REGION Network 4: Call production data cycle timer
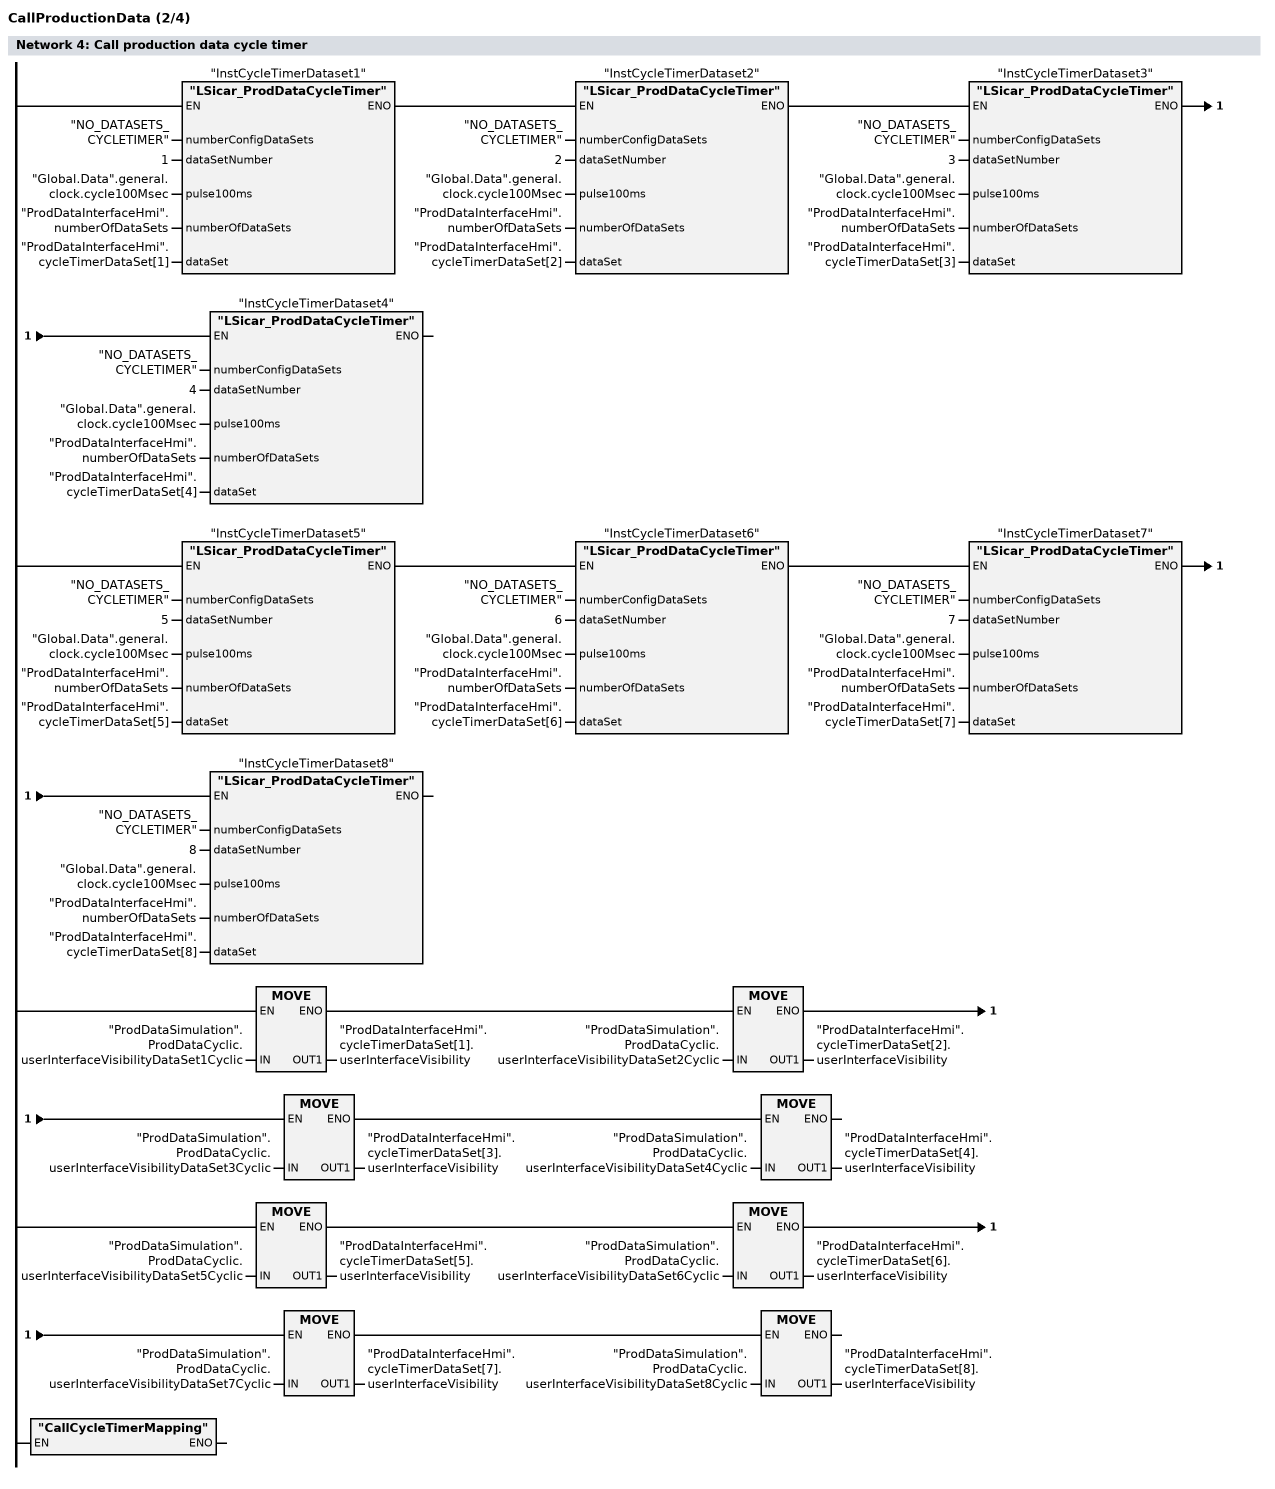
   RUNG wire#powerrail
      "InstCycleTimerDataset1"(numberConfigDataSets := "NO_DATASETS_CYCLETIMER", dataSetNumber := 1, pulse100ms := "Global.Data".general.clock.cycle100Msec, numberOfDataSets := "ProdDataInterfaceHmi".numberOfDataSets, dataSet := "ProdDataInterfaceHmi".cycleTimerDataSet[1])
      "InstCycleTimerDataset2"(numberConfigDataSets := "NO_DATASETS_CYCLETIMER", dataSetNumber := 2, pulse100ms := "Global.Data".general.clock.cycle100Msec, numberOfDataSets := "ProdDataInterfaceHmi".numberOfDataSets, dataSet := "ProdDataInterfaceHmi".cycleTimerDataSet[2])
      "InstCycleTimerDataset3"(numberConfigDataSets := "NO_DATASETS_CYCLETIMER", dataSetNumber := 3, pulse100ms := "Global.Data".general.clock.cycle100Msec, numberOfDataSets := "ProdDataInterfaceHmi".numberOfDataSets, dataSet := "ProdDataInterfaceHmi".cycleTimerDataSet[3])
      "InstCycleTimerDataset4"(numberConfigDataSets := "NO_DATASETS_CYCLETIMER", dataSetNumber := 4, pulse100ms := "Global.Data".general.clock.cycle100Msec, numberOfDataSets := "ProdDataInterfaceHmi".numberOfDataSets, dataSet := "ProdDataInterfaceHmi".cycleTimerDataSet[4])
   END_RUNG
   RUNG wire#powerrail
      "InstCycleTimerDataset5"(numberConfigDataSets := "NO_DATASETS_CYCLETIMER", dataSetNumber := 5, pulse100ms := "Global.Data".general.clock.cycle100Msec, numberOfDataSets := "ProdDataInterfaceHmi".numberOfDataSets, dataSet := "ProdDataInterfaceHmi".cycleTimerDataSet[5])
      "InstCycleTimerDataset6"(numberConfigDataSets := "NO_DATASETS_CYCLETIMER", dataSetNumber := 6, pulse100ms := "Global.Data".general.clock.cycle100Msec, numberOfDataSets := "ProdDataInterfaceHmi".numberOfDataSets, dataSet := "ProdDataInterfaceHmi".cycleTimerDataSet[6])
      "InstCycleTimerDataset7"(numberConfigDataSets := "NO_DATASETS_CYCLETIMER", dataSetNumber := 7, pulse100ms := "Global.Data".general.clock.cycle100Msec, numberOfDataSets := "ProdDataInterfaceHmi".numberOfDataSets, dataSet := "ProdDataInterfaceHmi".cycleTimerDataSet[7])
      "InstCycleTimerDataset8"(numberConfigDataSets := "NO_DATASETS_CYCLETIMER", dataSetNumber := 8, pulse100ms := "Global.Data".general.clock.cycle100Msec, numberOfDataSets := "ProdDataInterfaceHmi".numberOfDataSets, dataSet := "ProdDataInterfaceHmi".cycleTimerDataSet[8])
   END_RUNG
   RUNG wire#powerrail
      Move(in := "ProdDataSimulation".ProdDataCyclic.userInterfaceVisibilityDataSet1Cyclic, out1 => "ProdDataInterfaceHmi".cycleTimerDataSet[1].userInterfaceVisibility)
      Move(in := "ProdDataSimulation".ProdDataCyclic.userInterfaceVisibilityDataSet2Cyclic, out1 => "ProdDataInterfaceHmi".cycleTimerDataSet[2].userInterfaceVisibility)
      Move(in := "ProdDataSimulation".ProdDataCyclic.userInterfaceVisibilityDataSet3Cyclic, out1 => "ProdDataInterfaceHmi".cycleTimerDataSet[3].userInterfaceVisibility)
      Move(in := "ProdDataSimulation".ProdDataCyclic.userInterfaceVisibilityDataSet4Cyclic, out1 => "ProdDataInterfaceHmi".cycleTimerDataSet[4].userInterfaceVisibility)
   END_RUNG
   RUNG wire#powerrail
      Move(in := "ProdDataSimulation".ProdDataCyclic.userInterfaceVisibilityDataSet5Cyclic, out1 => "ProdDataInterfaceHmi".cycleTimerDataSet[5].userInterfaceVisibility)
      Move(in := "ProdDataSimulation".ProdDataCyclic.userInterfaceVisibilityDataSet6Cyclic, out1 => "ProdDataInterfaceHmi".cycleTimerDataSet[6].userInterfaceVisibility)
      Move(in := "ProdDataSimulation".ProdDataCyclic.userInterfaceVisibilityDataSet7Cyclic, out1 => "ProdDataInterfaceHmi".cycleTimerDataSet[7].userInterfaceVisibility)
      Move(in := "ProdDataSimulation".ProdDataCyclic.userInterfaceVisibilityDataSet8Cyclic, out1 => "ProdDataInterfaceHmi".cycleTimerDataSet[8].userInterfaceVisibility)
   END_RUNG
   RUNG wire#powerrail
      "CallCycleTimerMapping"()
   END_RUNG
   // the same network as SCL:
   "InstCycleTimerDataset1"(numberConfigDataSets := "NO_DATASETS_CYCLETIMER",   // "LSicar_ProdDataCycleTimer"
                           dataSetNumber := 1,
                           pulse100ms := "Global.Data".general.clock.cycle100Msec,
                           numberOfDataSets := "ProdDataInterfaceHmi".numberOfDataSets,
                           dataSet := "ProdDataInterfaceHmi".cycleTimerDataSet[1],
                           ENO => #_w1);
   "InstCycleTimerDataset2"(EN := #_w1,   // "LSicar_ProdDataCycleTimer"
                           numberConfigDataSets := "NO_DATASETS_CYCLETIMER",
                           dataSetNumber := 2,
                           pulse100ms := "Global.Data".general.clock.cycle100Msec,
                           numberOfDataSets := "ProdDataInterfaceHmi".numberOfDataSets,
                           dataSet := "ProdDataInterfaceHmi".cycleTimerDataSet[2],
                           ENO => #_w2);
   "InstCycleTimerDataset3"(EN := #_w2,   // "LSicar_ProdDataCycleTimer"
                           numberConfigDataSets := "NO_DATASETS_CYCLETIMER",
                           dataSetNumber := 3,
                           pulse100ms := "Global.Data".general.clock.cycle100Msec,
                           numberOfDataSets := "ProdDataInterfaceHmi".numberOfDataSets,
                           dataSet := "ProdDataInterfaceHmi".cycleTimerDataSet[3],
                           ENO => #_w3);
   IF #_w3 THEN
       "InstCycleTimerDataset4"(numberConfigDataSets := "NO_DATASETS_CYCLETIMER",   // "LSicar_ProdDataCycleTimer"
                               dataSetNumber := 4,
                               pulse100ms := "Global.Data".general.clock.cycle100Msec,
                               numberOfDataSets := "ProdDataInterfaceHmi".numberOfDataSets,
                               dataSet := "ProdDataInterfaceHmi".cycleTimerDataSet[4]);
   END_IF;
   "InstCycleTimerDataset5"(numberConfigDataSets := "NO_DATASETS_CYCLETIMER",   // "LSicar_ProdDataCycleTimer"
                           dataSetNumber := 5,
                           pulse100ms := "Global.Data".general.clock.cycle100Msec,
                           numberOfDataSets := "ProdDataInterfaceHmi".numberOfDataSets,
                           dataSet := "ProdDataInterfaceHmi".cycleTimerDataSet[5],
                           ENO => #_w4);
   "InstCycleTimerDataset6"(EN := #_w4,   // "LSicar_ProdDataCycleTimer"
                           numberConfigDataSets := "NO_DATASETS_CYCLETIMER",
                           dataSetNumber := 6,
                           pulse100ms := "Global.Data".general.clock.cycle100Msec,
                           numberOfDataSets := "ProdDataInterfaceHmi".numberOfDataSets,
                           dataSet := "ProdDataInterfaceHmi".cycleTimerDataSet[6],
                           ENO => #_w5);
   "InstCycleTimerDataset7"(EN := #_w5,   // "LSicar_ProdDataCycleTimer"
                           numberConfigDataSets := "NO_DATASETS_CYCLETIMER",
                           dataSetNumber := 7,
                           pulse100ms := "Global.Data".general.clock.cycle100Msec,
                           numberOfDataSets := "ProdDataInterfaceHmi".numberOfDataSets,
                           dataSet := "ProdDataInterfaceHmi".cycleTimerDataSet[7],
                           ENO => #_w6);
   IF #_w6 THEN
       "InstCycleTimerDataset8"(numberConfigDataSets := "NO_DATASETS_CYCLETIMER",   // "LSicar_ProdDataCycleTimer"
                               dataSetNumber := 8,
                               pulse100ms := "Global.Data".general.clock.cycle100Msec,
                               numberOfDataSets := "ProdDataInterfaceHmi".numberOfDataSets,
                               dataSet := "ProdDataInterfaceHmi".cycleTimerDataSet[8]);
   END_IF;
   "ProdDataInterfaceHmi".cycleTimerDataSet[1].userInterfaceVisibility := "ProdDataSimulation".ProdDataCyclic.userInterfaceVisibilityDataSet1Cyclic;
   "ProdDataInterfaceHmi".cycleTimerDataSet[2].userInterfaceVisibility := "ProdDataSimulation".ProdDataCyclic.userInterfaceVisibilityDataSet2Cyclic;
   "ProdDataInterfaceHmi".cycleTimerDataSet[3].userInterfaceVisibility := "ProdDataSimulation".ProdDataCyclic.userInterfaceVisibilityDataSet3Cyclic;
   "ProdDataInterfaceHmi".cycleTimerDataSet[4].userInterfaceVisibility := "ProdDataSimulation".ProdDataCyclic.userInterfaceVisibilityDataSet4Cyclic;
   "ProdDataInterfaceHmi".cycleTimerDataSet[5].userInterfaceVisibility := "ProdDataSimulation".ProdDataCyclic.userInterfaceVisibilityDataSet5Cyclic;
   "ProdDataInterfaceHmi".cycleTimerDataSet[6].userInterfaceVisibility := "ProdDataSimulation".ProdDataCyclic.userInterfaceVisibilityDataSet6Cyclic;
   "ProdDataInterfaceHmi".cycleTimerDataSet[7].userInterfaceVisibility := "ProdDataSimulation".ProdDataCyclic.userInterfaceVisibilityDataSet7Cyclic;
   "ProdDataInterfaceHmi".cycleTimerDataSet[8].userInterfaceVisibility := "ProdDataSimulation".ProdDataCyclic.userInterfaceVisibilityDataSet8Cyclic;
   "CallCycleTimerMapping"();
END_REGION

REGION Network 5: Beispiel: Limit Value 1..2 / Call production data limit values
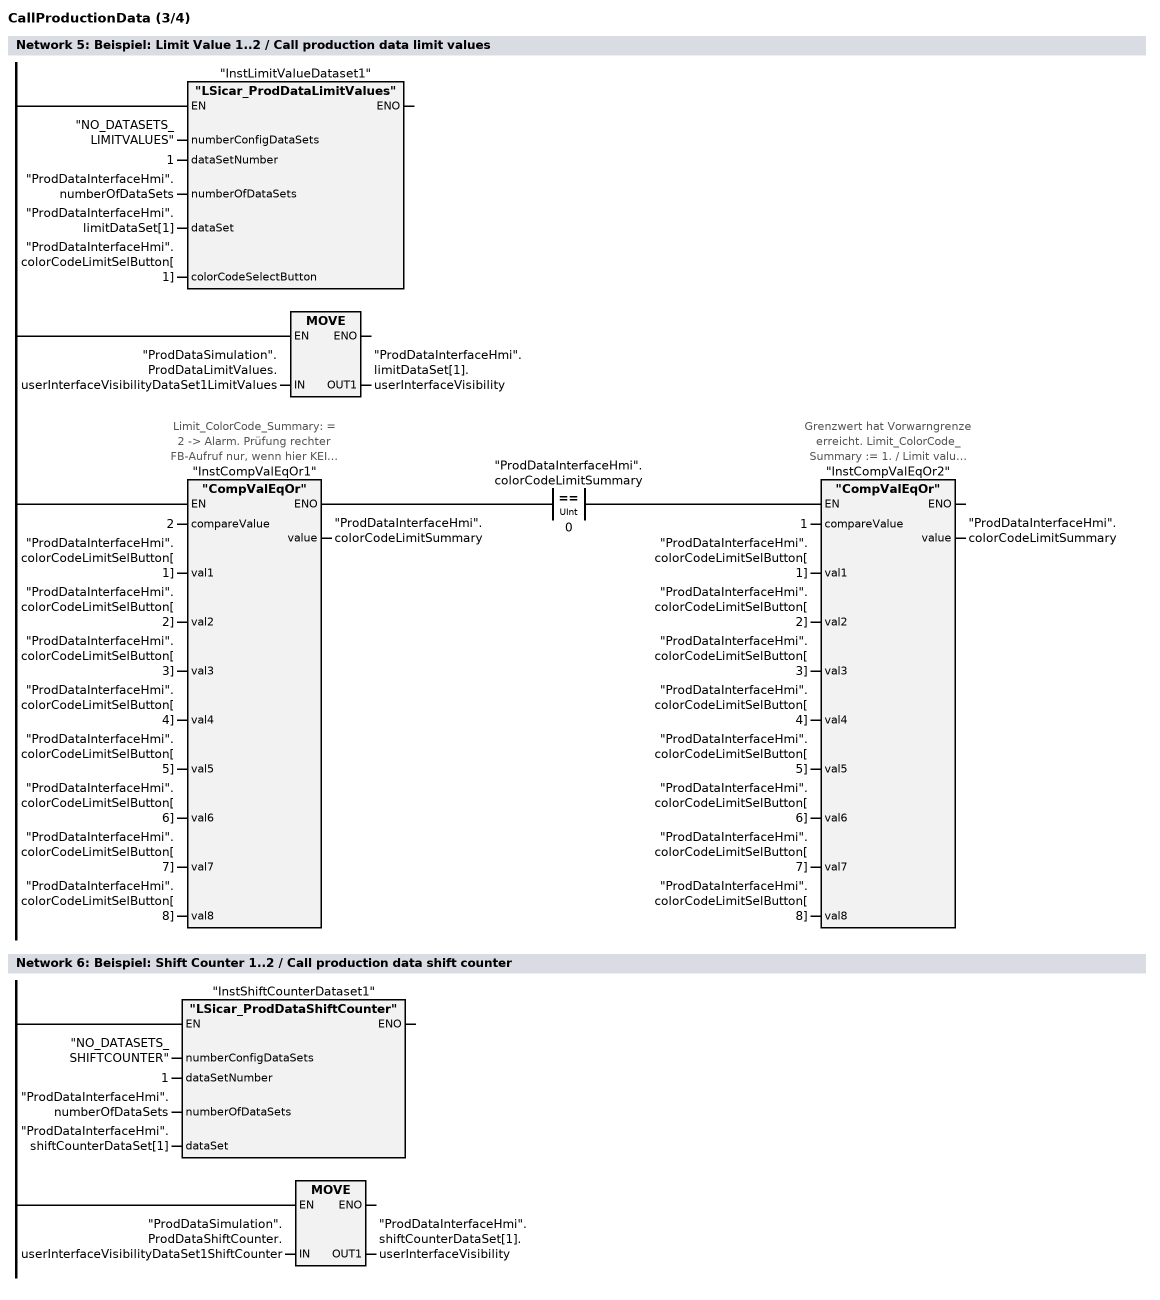
   RUNG wire#powerrail
      "InstLimitValueDataset1"(numberConfigDataSets := "NO_DATASETS_LIMITVALUES", dataSetNumber := 1, numberOfDataSets := "ProdDataInterfaceHmi".numberOfDataSets, dataSet := "ProdDataInterfaceHmi".limitDataSet[1], colorCodeSelectButton := "ProdDataInterfaceHmi".colorCodeLimitSelButton[1])
   END_RUNG
   RUNG wire#powerrail
      Move(in := "ProdDataSimulation".ProdDataLimitValues.userInterfaceVisibilityDataSet1LimitValues, out1 => "ProdDataInterfaceHmi".limitDataSet[1].userInterfaceVisibility)
   END_RUNG
   RUNG wire#powerrail
      "InstCompValEqOr1"(compareValue := 2, val1 := "ProdDataInterfaceHmi".colorCodeLimitSelButton[1], val2 := "ProdDataInterfaceHmi".colorCodeLimitSelButton[2], val3 := "ProdDataInterfaceHmi".colorCodeLimitSelButton[3], val4 := "ProdDataInterfaceHmi".colorCodeLimitSelButton[4], val5 := "ProdDataInterfaceHmi".colorCodeLimitSelButton[5], val6 := "ProdDataInterfaceHmi".colorCodeLimitSelButton[6], val7 := "ProdDataInterfaceHmi".colorCodeLimitSelButton[7], val8 := "ProdDataInterfaceHmi".colorCodeLimitSelButton[8], value => "ProdDataInterfaceHmi".colorCodeLimitSummary)   // Limit_ColorCode_Summary: = 2 -> Alarm. Prüfung rechter FB-Aufruf nur, wenn hier KEIN Alarm (VALUE = 0) ansteht; Alarm ist höher prior. / Limit value = 2 -> Alarm. Limit_ColorCode_Summary := 2. Call right block only, if NO alarm (VALUE = 0) is pending here; alarm is higher prior.
      { S7_Templates := "SrcType := UInt" } EQ_Contact(in1 := "ProdDataInterfaceHmi".colorCodeLimitSummary, in2 := 0)
      "InstCompValEqOr2"(compareValue := 1, val1 := "ProdDataInterfaceHmi".colorCodeLimitSelButton[1], val2 := "ProdDataInterfaceHmi".colorCodeLimitSelButton[2], val3 := "ProdDataInterfaceHmi".colorCodeLimitSelButton[3], val4 := "ProdDataInterfaceHmi".colorCodeLimitSelButton[4], val5 := "ProdDataInterfaceHmi".colorCodeLimitSelButton[5], val6 := "ProdDataInterfaceHmi".colorCodeLimitSelButton[6], val7 := "ProdDataInterfaceHmi".colorCodeLimitSelButton[7], val8 := "ProdDataInterfaceHmi".colorCodeLimitSelButton[8], value => "ProdDataInterfaceHmi".colorCodeLimitSummary)   // Grenzwert hat Vorwarngrenze erreicht. Limit_ColorCode_Summary := 1. / Limit value <= Prewarn value. Limit_ColorCode_Summary := 1.
   END_RUNG
   // the same network as SCL:
   "InstLimitValueDataset1"(numberConfigDataSets := "NO_DATASETS_LIMITVALUES",   // "LSicar_ProdDataLimitValues"
                           dataSetNumber := 1,
                           numberOfDataSets := "ProdDataInterfaceHmi".numberOfDataSets,
                           dataSet := "ProdDataInterfaceHmi".limitDataSet[1],
                           colorCodeSelectButton := "ProdDataInterfaceHmi".colorCodeLimitSelButton[1]);
   "ProdDataInterfaceHmi".limitDataSet[1].userInterfaceVisibility := "ProdDataSimulation".ProdDataLimitValues.userInterfaceVisibilityDataSet1LimitValues;
   "InstCompValEqOr1"(compareValue := 2,   // "CompValEqOr": Limit_ColorCode_Summary: = 2 -> Alarm. Prüfung rechter FB-Aufruf nur, wenn hier KEIN Alarm (VALUE = 0) ansteht; Alarm ist höher prior. / Limit value = 2 -> Alarm. Limit_ColorCode_Summary := 2. Call right block only, if NO alarm (VALUE = 0) is pending here; alarm is higher prior.
                      val1 := "ProdDataInterfaceHmi".colorCodeLimitSelButton[1],
                      val2 := "ProdDataInterfaceHmi".colorCodeLimitSelButton[2],
                      val3 := "ProdDataInterfaceHmi".colorCodeLimitSelButton[3],
                      val4 := "ProdDataInterfaceHmi".colorCodeLimitSelButton[4],
                      val5 := "ProdDataInterfaceHmi".colorCodeLimitSelButton[5],
                      val6 := "ProdDataInterfaceHmi".colorCodeLimitSelButton[6],
                      val7 := "ProdDataInterfaceHmi".colorCodeLimitSelButton[7],
                      val8 := "ProdDataInterfaceHmi".colorCodeLimitSelButton[8],
                      value => "ProdDataInterfaceHmi".colorCodeLimitSummary,
                      ENO => #_w1);
   IF #_w1 AND ("ProdDataInterfaceHmi".colorCodeLimitSummary = 0) THEN
       "InstCompValEqOr2"(compareValue := 1,   // "CompValEqOr": Grenzwert hat Vorwarngrenze erreicht. Limit_ColorCode_Summary := 1. / Limit value <= Prewarn value. Limit_ColorCode_Summary := 1.
                          val1 := "ProdDataInterfaceHmi".colorCodeLimitSelButton[1],
                          val2 := "ProdDataInterfaceHmi".colorCodeLimitSelButton[2],
                          val3 := "ProdDataInterfaceHmi".colorCodeLimitSelButton[3],
                          val4 := "ProdDataInterfaceHmi".colorCodeLimitSelButton[4],
                          val5 := "ProdDataInterfaceHmi".colorCodeLimitSelButton[5],
                          val6 := "ProdDataInterfaceHmi".colorCodeLimitSelButton[6],
                          val7 := "ProdDataInterfaceHmi".colorCodeLimitSelButton[7],
                          val8 := "ProdDataInterfaceHmi".colorCodeLimitSelButton[8],
                          value => "ProdDataInterfaceHmi".colorCodeLimitSummary);
   END_IF;
END_REGION

REGION Network 6: Beispiel: Shift Counter 1..2 / Call production data shift counter
   RUNG wire#powerrail
      "InstShiftCounterDataset1"(numberConfigDataSets := "NO_DATASETS_SHIFTCOUNTER", dataSetNumber := 1, numberOfDataSets := "ProdDataInterfaceHmi".numberOfDataSets, dataSet := "ProdDataInterfaceHmi".shiftCounterDataSet[1])
   END_RUNG
   RUNG wire#powerrail
      Move(in := "ProdDataSimulation".ProdDataShiftCounter.userInterfaceVisibilityDataSet1ShiftCounter, out1 => "ProdDataInterfaceHmi".shiftCounterDataSet[1].userInterfaceVisibility)
   END_RUNG
   // the same network as SCL:
   "InstShiftCounterDataset1"(numberConfigDataSets := "NO_DATASETS_SHIFTCOUNTER",   // "LSicar_ProdDataShiftCounter"
                           dataSetNumber := 1,
                           numberOfDataSets := "ProdDataInterfaceHmi".numberOfDataSets,
                           dataSet := "ProdDataInterfaceHmi".shiftCounterDataSet[1]);
   "ProdDataInterfaceHmi".shiftCounterDataSet[1].userInterfaceVisibility := "ProdDataSimulation".ProdDataShiftCounter.userInterfaceVisibilityDataSet1ShiftCounter;
END_REGION

REGION Network 7: Beispiel Schichtproduktions-Zeiten / Call shift production times
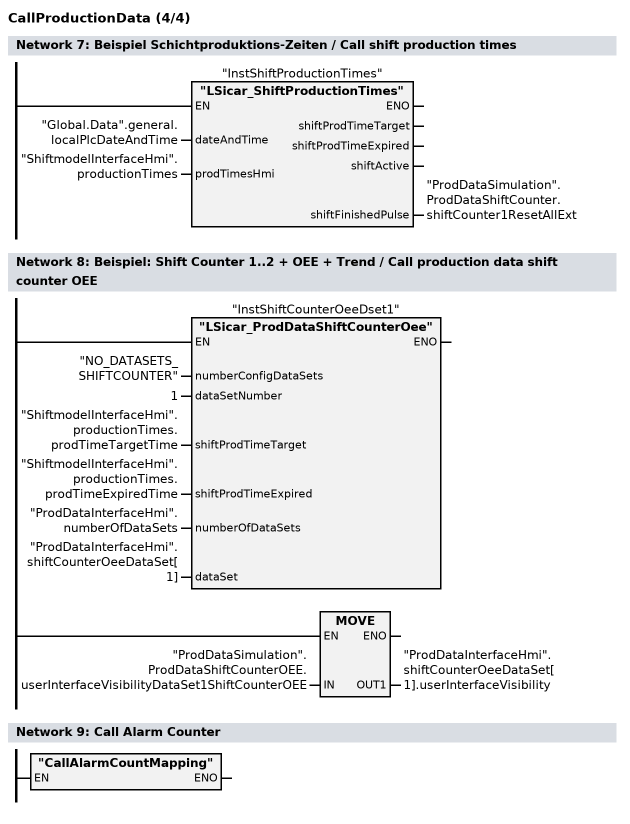
   RUNG wire#powerrail
      "InstShiftProductionTimes"(dateAndTime := "Global.Data".general.localPlcDateAndTime, prodTimesHmi := "ShiftmodelInterfaceHmi".productionTimes, shiftProdTimeTarget =>, shiftProdTimeExpired =>, shiftActive =>, shiftFinishedPulse => "ProdDataSimulation".ProdDataShiftCounter.shiftCounter1ResetAllExt)
   END_RUNG
   // the same network as SCL:
   "InstShiftProductionTimes"(dateAndTime := "Global.Data".general.localPlcDateAndTime,   // "LSicar_ShiftProductionTimes"
                           prodTimesHmi := "ShiftmodelInterfaceHmi".productionTimes,
                           shiftFinishedPulse => "ProdDataSimulation".ProdDataShiftCounter.shiftCounter1ResetAllExt);
END_REGION

REGION Network 8: Beispiel: Shift Counter 1..2 + OEE + Trend / Call production data shift counter OEE
   RUNG wire#powerrail
      "InstShiftCounterOeeDset1"(numberConfigDataSets := "NO_DATASETS_SHIFTCOUNTER", dataSetNumber := 1, shiftProdTimeTarget := "ShiftmodelInterfaceHmi".productionTimes.prodTimeTargetTime, shiftProdTimeExpired := "ShiftmodelInterfaceHmi".productionTimes.prodTimeExpiredTime, numberOfDataSets := "ProdDataInterfaceHmi".numberOfDataSets, dataSet := "ProdDataInterfaceHmi".shiftCounterOeeDataSet[1])
   END_RUNG
   RUNG wire#powerrail
      Move(in := "ProdDataSimulation".ProdDataShiftCounterOEE.userInterfaceVisibilityDataSet1ShiftCounterOEE, out1 => "ProdDataInterfaceHmi".shiftCounterOeeDataSet[1].userInterfaceVisibility)
   END_RUNG
   // the same network as SCL:
   "InstShiftCounterOeeDset1"(numberConfigDataSets := "NO_DATASETS_SHIFTCOUNTER",   // "LSicar_ProdDataShiftCounterOee"
                           dataSetNumber := 1,
                           shiftProdTimeTarget := "ShiftmodelInterfaceHmi".productionTimes.prodTimeTargetTime,
                           shiftProdTimeExpired := "ShiftmodelInterfaceHmi".productionTimes.prodTimeExpiredTime,
                           numberOfDataSets := "ProdDataInterfaceHmi".numberOfDataSets,
                           dataSet := "ProdDataInterfaceHmi".shiftCounterOeeDataSet[1]);
   "ProdDataInterfaceHmi".shiftCounterOeeDataSet[1].userInterfaceVisibility := "ProdDataSimulation".ProdDataShiftCounterOEE.userInterfaceVisibilityDataSet1ShiftCounterOEE;
END_REGION

REGION Network 9: Call Alarm Counter
   RUNG wire#powerrail
      "CallAlarmCountMapping"()
   END_RUNG
   // the same network as SCL:
   "CallAlarmCountMapping"();
END_REGION
END_FUNCTION

FUNCTION "CallCounterMapping" : Void   // FC94, LAD
// stored: SetENOAutomatically false
   VAR CONSTANT
      TRUE : Bool := TRUE;
   END_VAR
BEGIN

REGION Network 1: Input Qty
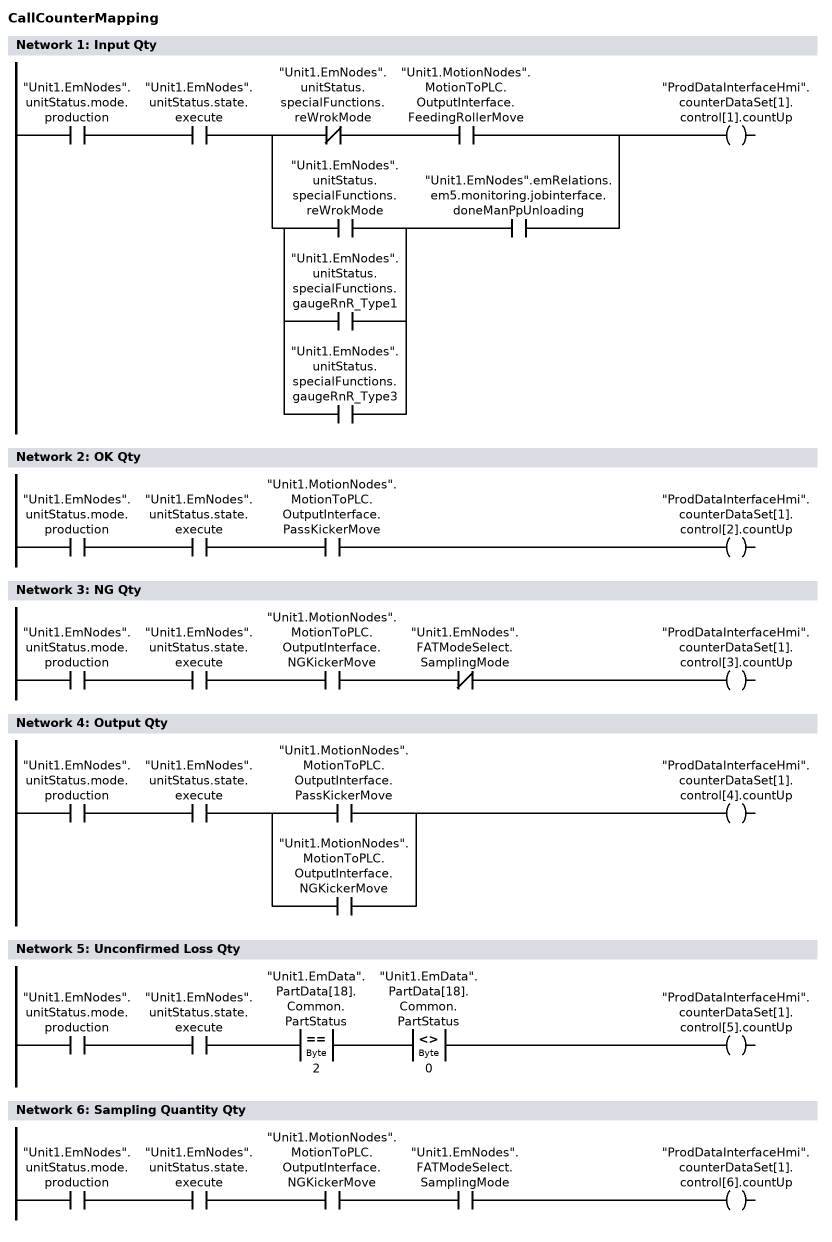
   RUNG wire#powerrail
      Contact( "Unit1.EmNodes".unitStatus.mode.production )
      Contact( "Unit1.EmNodes".unitStatus.state.execute )
      wire#w1
      I_Contact( "Unit1.EmNodes".unitStatus.specialFunctions.reWrokMode )
      Contact( "Unit1.MotionNodes".MotionToPLC.OutputInterface.FeedingRollerMove )
      wire#w2
      Coil( "ProdDataInterfaceHmi".counterDataSet[1].control[1].countUp )
   END_RUNG
   RUNG wire#w1
      Contact( "Unit1.EmNodes".unitStatus.specialFunctions.reWrokMode )
      wire#w3
      Contact( "Unit1.EmNodes".emRelations.em5.monitoring.jobinterface.doneManPpUnloading )
   END_RUNG wire#w2
   RUNG wire#w1
      Contact( "Unit1.EmNodes".unitStatus.specialFunctions.gaugeRnR_Type1 )
   END_RUNG wire#w3
   RUNG wire#w1
      Contact( "Unit1.EmNodes".unitStatus.specialFunctions.gaugeRnR_Type3 )
   END_RUNG wire#w3
   // the same network as SCL:
   "ProdDataInterfaceHmi".counterDataSet[1].control[1].countUp := "Unit1.EmNodes".unitStatus.mode.production AND "Unit1.EmNodes".unitStatus.state.execute AND ((NOT "Unit1.EmNodes".unitStatus.specialFunctions.reWrokMode AND "Unit1.MotionNodes".MotionToPLC.OutputInterface.FeedingRollerMove) OR (("Unit1.EmNodes".unitStatus.specialFunctions.reWrokMode OR "Unit1.EmNodes".unitStatus.specialFunctions.gaugeRnR_Type1 OR "Unit1.EmNodes".unitStatus.specialFunctions.gaugeRnR_Type3) AND "Unit1.EmNodes".emRelations.em5.monitoring.jobinterface.doneManPpUnloading));
END_REGION

REGION Network 2: OK Qty
   RUNG wire#powerrail
      Contact( "Unit1.EmNodes".unitStatus.mode.production )
      Contact( "Unit1.EmNodes".unitStatus.state.execute )
      Contact( "Unit1.MotionNodes".MotionToPLC.OutputInterface.PassKickerMove )
      Coil( "ProdDataInterfaceHmi".counterDataSet[1].control[2].countUp )
   END_RUNG
   // the same network as SCL:
   "ProdDataInterfaceHmi".counterDataSet[1].control[2].countUp := "Unit1.EmNodes".unitStatus.mode.production AND "Unit1.EmNodes".unitStatus.state.execute AND "Unit1.MotionNodes".MotionToPLC.OutputInterface.PassKickerMove;
END_REGION

REGION Network 3: NG Qty
   RUNG wire#powerrail
      Contact( "Unit1.EmNodes".unitStatus.mode.production )
      Contact( "Unit1.EmNodes".unitStatus.state.execute )
      Contact( "Unit1.MotionNodes".MotionToPLC.OutputInterface.NGKickerMove )
      I_Contact( "Unit1.EmNodes".FATModeSelect.SamplingMode )
      Coil( "ProdDataInterfaceHmi".counterDataSet[1].control[3].countUp )
   END_RUNG
   // the same network as SCL:
   "ProdDataInterfaceHmi".counterDataSet[1].control[3].countUp := "Unit1.EmNodes".unitStatus.mode.production AND "Unit1.EmNodes".unitStatus.state.execute AND "Unit1.MotionNodes".MotionToPLC.OutputInterface.NGKickerMove AND NOT "Unit1.EmNodes".FATModeSelect.SamplingMode;
END_REGION

REGION Network 4: Output Qty
   RUNG wire#powerrail
      Contact( "Unit1.EmNodes".unitStatus.mode.production )
      Contact( "Unit1.EmNodes".unitStatus.state.execute )
      wire#w1
      Contact( "Unit1.MotionNodes".MotionToPLC.OutputInterface.PassKickerMove )
      wire#w2
      Coil( "ProdDataInterfaceHmi".counterDataSet[1].control[4].countUp )
   END_RUNG
   RUNG wire#w1
      Contact( "Unit1.MotionNodes".MotionToPLC.OutputInterface.NGKickerMove )
   END_RUNG wire#w2
   // the same network as SCL:
   "ProdDataInterfaceHmi".counterDataSet[1].control[4].countUp := "Unit1.EmNodes".unitStatus.mode.production AND "Unit1.EmNodes".unitStatus.state.execute AND ("Unit1.MotionNodes".MotionToPLC.OutputInterface.PassKickerMove OR "Unit1.MotionNodes".MotionToPLC.OutputInterface.NGKickerMove);
END_REGION

REGION Network 5: Unconfirmed Loss Qty
   RUNG wire#powerrail
      Contact( "Unit1.EmNodes".unitStatus.mode.production )
      Contact( "Unit1.EmNodes".unitStatus.state.execute )
      { S7_Templates := "SrcType := Byte" } EQ_Contact(in1 := "Unit1.EmData".PartData[18].Common.PartStatus, in2 := 2)
      { S7_Templates := "SrcType := Byte" } NE_Contact(in1 := "Unit1.EmData".PartData[18].Common.PartStatus, in2 := 0)
      Coil( "ProdDataInterfaceHmi".counterDataSet[1].control[5].countUp )
   END_RUNG
   // the same network as SCL:
   "ProdDataInterfaceHmi".counterDataSet[1].control[5].countUp := "Unit1.EmNodes".unitStatus.mode.production AND "Unit1.EmNodes".unitStatus.state.execute AND ("Unit1.EmData".PartData[18].Common.PartStatus = 2) AND ("Unit1.EmData".PartData[18].Common.PartStatus <> 0);
END_REGION

REGION Network 6: Sampling Quantity Qty
   RUNG wire#powerrail
      Contact( "Unit1.EmNodes".unitStatus.mode.production )
      Contact( "Unit1.EmNodes".unitStatus.state.execute )
      Contact( "Unit1.MotionNodes".MotionToPLC.OutputInterface.NGKickerMove )
      Contact( "Unit1.EmNodes".FATModeSelect.SamplingMode )
      Coil( "ProdDataInterfaceHmi".counterDataSet[1].control[6].countUp )
   END_RUNG
   // the same network as SCL:
   "ProdDataInterfaceHmi".counterDataSet[1].control[6].countUp := "Unit1.EmNodes".unitStatus.mode.production AND "Unit1.EmNodes".unitStatus.state.execute AND "Unit1.MotionNodes".MotionToPLC.OutputInterface.NGKickerMove AND "Unit1.EmNodes".FATModeSelect.SamplingMode;
END_REGION
END_FUNCTION

FUNCTION "CallCycleTimerMapping" : Void   // FC4, LAD
// stored: SetENOAutomatically false
   VAR CONSTANT
      TRUE : Bool := TRUE;
   END_VAR
BEGIN

REGION Network 1: cycleTimerDataSet[1]
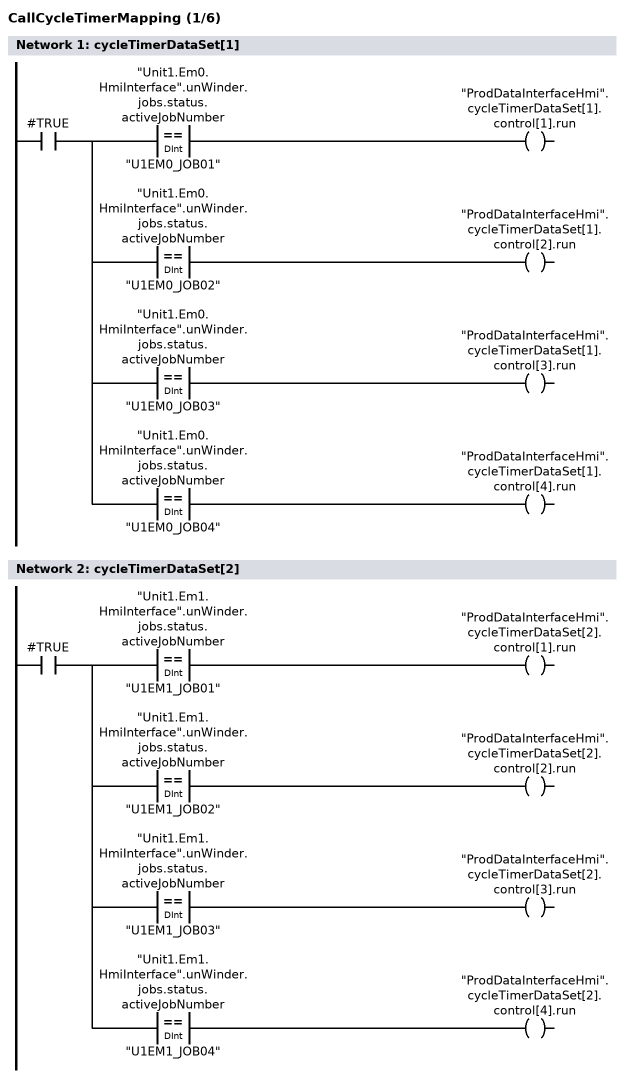
   RUNG wire#powerrail
      Contact( #TRUE )
      wire#w1
      { S7_Templates := "SrcType := DInt" } EQ_Contact(in1 := "Unit1.Em0.HmiInterface".unWinder.jobs.status.activeJobNumber, in2 := "U1EM0_JOB01")
      Coil( "ProdDataInterfaceHmi".cycleTimerDataSet[1].control[1].run )
   END_RUNG
   RUNG wire#w1
      { S7_Templates := "SrcType := DInt" } EQ_Contact(in1 := "Unit1.Em0.HmiInterface".unWinder.jobs.status.activeJobNumber, in2 := "U1EM0_JOB02")
      Coil( "ProdDataInterfaceHmi".cycleTimerDataSet[1].control[2].run )
   END_RUNG
   RUNG wire#w1
      { S7_Templates := "SrcType := DInt" } EQ_Contact(in1 := "Unit1.Em0.HmiInterface".unWinder.jobs.status.activeJobNumber, in2 := "U1EM0_JOB03")
      Coil( "ProdDataInterfaceHmi".cycleTimerDataSet[1].control[3].run )
   END_RUNG
   RUNG wire#w1
      { S7_Templates := "SrcType := DInt" } EQ_Contact(in1 := "Unit1.Em0.HmiInterface".unWinder.jobs.status.activeJobNumber, in2 := "U1EM0_JOB04")
      Coil( "ProdDataInterfaceHmi".cycleTimerDataSet[1].control[4].run )
   END_RUNG
   // the same network as SCL:
   "ProdDataInterfaceHmi".cycleTimerDataSet[1].control[1].run := #TRUE AND ("Unit1.Em0.HmiInterface".unWinder.jobs.status.activeJobNumber = "U1EM0_JOB01");
   "ProdDataInterfaceHmi".cycleTimerDataSet[1].control[2].run := #TRUE AND ("Unit1.Em0.HmiInterface".unWinder.jobs.status.activeJobNumber = "U1EM0_JOB02");
   "ProdDataInterfaceHmi".cycleTimerDataSet[1].control[3].run := #TRUE AND ("Unit1.Em0.HmiInterface".unWinder.jobs.status.activeJobNumber = "U1EM0_JOB03");
   "ProdDataInterfaceHmi".cycleTimerDataSet[1].control[4].run := #TRUE AND ("Unit1.Em0.HmiInterface".unWinder.jobs.status.activeJobNumber = "U1EM0_JOB04");
END_REGION

REGION Network 2: cycleTimerDataSet[2]
   RUNG wire#powerrail
      Contact( #TRUE )
      wire#w1
      { S7_Templates := "SrcType := DInt" } EQ_Contact(in1 := "Unit1.Em1.HmiInterface".unWinder.jobs.status.activeJobNumber, in2 := "U1EM1_JOB01")
      Coil( "ProdDataInterfaceHmi".cycleTimerDataSet[2].control[1].run )
   END_RUNG
   RUNG wire#w1
      { S7_Templates := "SrcType := DInt" } EQ_Contact(in1 := "Unit1.Em1.HmiInterface".unWinder.jobs.status.activeJobNumber, in2 := "U1EM1_JOB02")
      Coil( "ProdDataInterfaceHmi".cycleTimerDataSet[2].control[2].run )
   END_RUNG
   RUNG wire#w1
      { S7_Templates := "SrcType := DInt" } EQ_Contact(in1 := "Unit1.Em1.HmiInterface".unWinder.jobs.status.activeJobNumber, in2 := "U1EM1_JOB03")
      Coil( "ProdDataInterfaceHmi".cycleTimerDataSet[2].control[3].run )
   END_RUNG
   RUNG wire#w1
      { S7_Templates := "SrcType := DInt" } EQ_Contact(in1 := "Unit1.Em1.HmiInterface".unWinder.jobs.status.activeJobNumber, in2 := "U1EM1_JOB04")
      Coil( "ProdDataInterfaceHmi".cycleTimerDataSet[2].control[4].run )
   END_RUNG
   // the same network as SCL:
   "ProdDataInterfaceHmi".cycleTimerDataSet[2].control[1].run := #TRUE AND ("Unit1.Em1.HmiInterface".unWinder.jobs.status.activeJobNumber = "U1EM1_JOB01");
   "ProdDataInterfaceHmi".cycleTimerDataSet[2].control[2].run := #TRUE AND ("Unit1.Em1.HmiInterface".unWinder.jobs.status.activeJobNumber = "U1EM1_JOB02");
   "ProdDataInterfaceHmi".cycleTimerDataSet[2].control[3].run := #TRUE AND ("Unit1.Em1.HmiInterface".unWinder.jobs.status.activeJobNumber = "U1EM1_JOB03");
   "ProdDataInterfaceHmi".cycleTimerDataSet[2].control[4].run := #TRUE AND ("Unit1.Em1.HmiInterface".unWinder.jobs.status.activeJobNumber = "U1EM1_JOB04");
END_REGION

REGION Network 3: cycleTimerDataSet[3]
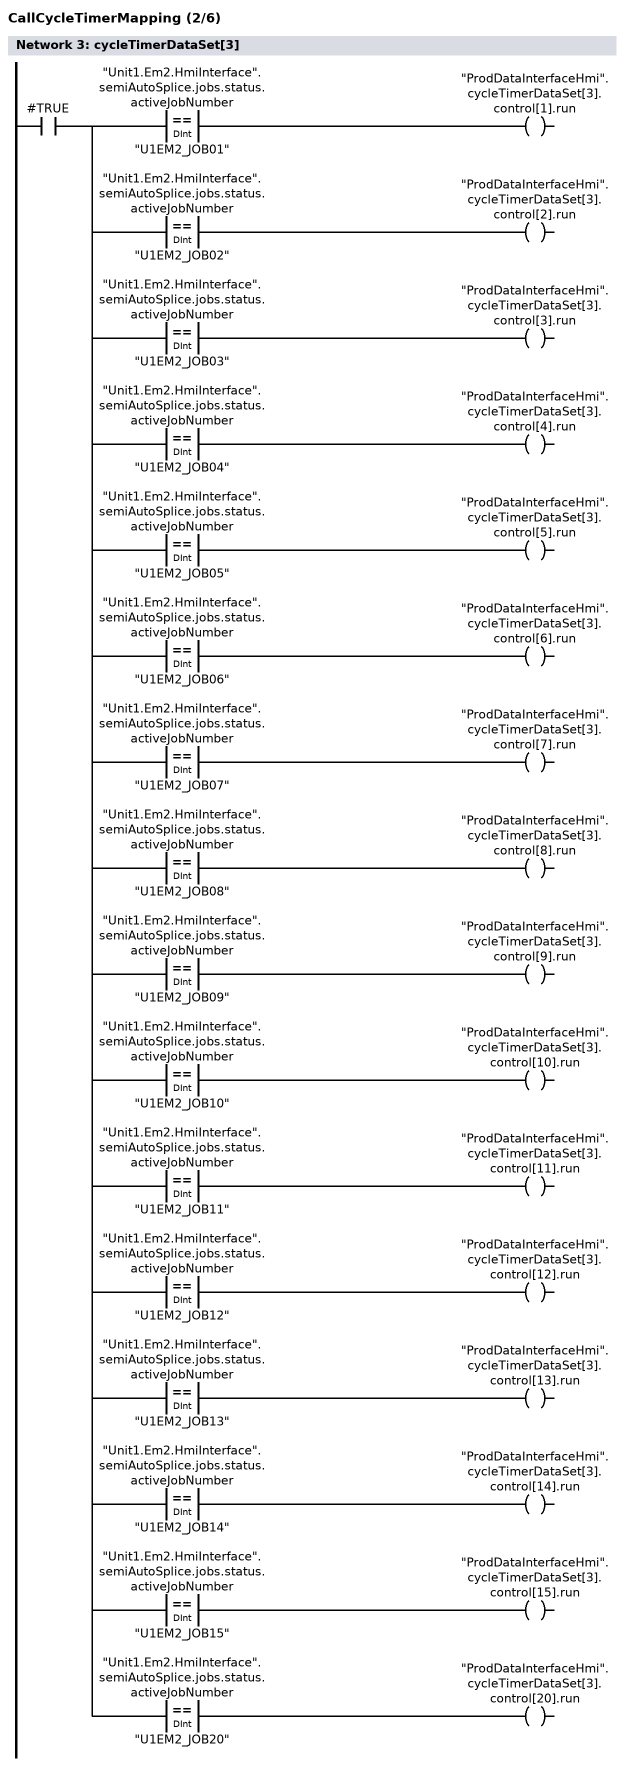
   RUNG wire#powerrail
      Contact( #TRUE )
      wire#w1
      { S7_Templates := "SrcType := DInt" } EQ_Contact(in1 := "Unit1.Em2.HmiInterface".semiAutoSplice.jobs.status.activeJobNumber, in2 := "U1EM2_JOB01")
      Coil( "ProdDataInterfaceHmi".cycleTimerDataSet[3].control[1].run )
   END_RUNG
   RUNG wire#w1
      { S7_Templates := "SrcType := DInt" } EQ_Contact(in1 := "Unit1.Em2.HmiInterface".semiAutoSplice.jobs.status.activeJobNumber, in2 := "U1EM2_JOB02")
      Coil( "ProdDataInterfaceHmi".cycleTimerDataSet[3].control[2].run )
   END_RUNG
   RUNG wire#w1
      { S7_Templates := "SrcType := DInt" } EQ_Contact(in1 := "Unit1.Em2.HmiInterface".semiAutoSplice.jobs.status.activeJobNumber, in2 := "U1EM2_JOB03")
      Coil( "ProdDataInterfaceHmi".cycleTimerDataSet[3].control[3].run )
   END_RUNG
   RUNG wire#w1
      { S7_Templates := "SrcType := DInt" } EQ_Contact(in1 := "Unit1.Em2.HmiInterface".semiAutoSplice.jobs.status.activeJobNumber, in2 := "U1EM2_JOB04")
      Coil( "ProdDataInterfaceHmi".cycleTimerDataSet[3].control[4].run )
   END_RUNG
   RUNG wire#w1
      { S7_Templates := "SrcType := DInt" } EQ_Contact(in1 := "Unit1.Em2.HmiInterface".semiAutoSplice.jobs.status.activeJobNumber, in2 := "U1EM2_JOB05")
      Coil( "ProdDataInterfaceHmi".cycleTimerDataSet[3].control[5].run )
   END_RUNG
   RUNG wire#w1
      { S7_Templates := "SrcType := DInt" } EQ_Contact(in1 := "Unit1.Em2.HmiInterface".semiAutoSplice.jobs.status.activeJobNumber, in2 := "U1EM2_JOB06")
      Coil( "ProdDataInterfaceHmi".cycleTimerDataSet[3].control[6].run )
   END_RUNG
   RUNG wire#w1
      { S7_Templates := "SrcType := DInt" } EQ_Contact(in1 := "Unit1.Em2.HmiInterface".semiAutoSplice.jobs.status.activeJobNumber, in2 := "U1EM2_JOB07")
      Coil( "ProdDataInterfaceHmi".cycleTimerDataSet[3].control[7].run )
   END_RUNG
   RUNG wire#w1
      { S7_Templates := "SrcType := DInt" } EQ_Contact(in1 := "Unit1.Em2.HmiInterface".semiAutoSplice.jobs.status.activeJobNumber, in2 := "U1EM2_JOB08")
      Coil( "ProdDataInterfaceHmi".cycleTimerDataSet[3].control[8].run )
   END_RUNG
   RUNG wire#w1
      { S7_Templates := "SrcType := DInt" } EQ_Contact(in1 := "Unit1.Em2.HmiInterface".semiAutoSplice.jobs.status.activeJobNumber, in2 := "U1EM2_JOB09")
      Coil( "ProdDataInterfaceHmi".cycleTimerDataSet[3].control[9].run )
   END_RUNG
   RUNG wire#w1
      { S7_Templates := "SrcType := DInt" } EQ_Contact(in1 := "Unit1.Em2.HmiInterface".semiAutoSplice.jobs.status.activeJobNumber, in2 := "U1EM2_JOB10")
      Coil( "ProdDataInterfaceHmi".cycleTimerDataSet[3].control[10].run )
   END_RUNG
   RUNG wire#w1
      { S7_Templates := "SrcType := DInt" } EQ_Contact(in1 := "Unit1.Em2.HmiInterface".semiAutoSplice.jobs.status.activeJobNumber, in2 := "U1EM2_JOB11")
      Coil( "ProdDataInterfaceHmi".cycleTimerDataSet[3].control[11].run )
   END_RUNG
   RUNG wire#w1
      { S7_Templates := "SrcType := DInt" } EQ_Contact(in1 := "Unit1.Em2.HmiInterface".semiAutoSplice.jobs.status.activeJobNumber, in2 := "U1EM2_JOB12")
      Coil( "ProdDataInterfaceHmi".cycleTimerDataSet[3].control[12].run )
   END_RUNG
   RUNG wire#w1
      { S7_Templates := "SrcType := DInt" } EQ_Contact(in1 := "Unit1.Em2.HmiInterface".semiAutoSplice.jobs.status.activeJobNumber, in2 := "U1EM2_JOB13")
      Coil( "ProdDataInterfaceHmi".cycleTimerDataSet[3].control[13].run )
   END_RUNG
   RUNG wire#w1
      { S7_Templates := "SrcType := DInt" } EQ_Contact(in1 := "Unit1.Em2.HmiInterface".semiAutoSplice.jobs.status.activeJobNumber, in2 := "U1EM2_JOB14")
      Coil( "ProdDataInterfaceHmi".cycleTimerDataSet[3].control[14].run )
   END_RUNG
   RUNG wire#w1
      { S7_Templates := "SrcType := DInt" } EQ_Contact(in1 := "Unit1.Em2.HmiInterface".semiAutoSplice.jobs.status.activeJobNumber, in2 := "U1EM2_JOB15")
      Coil( "ProdDataInterfaceHmi".cycleTimerDataSet[3].control[15].run )
   END_RUNG
   RUNG wire#w1
      { S7_Templates := "SrcType := DInt" } EQ_Contact(in1 := "Unit1.Em2.HmiInterface".semiAutoSplice.jobs.status.activeJobNumber, in2 := "U1EM2_JOB20")
      Coil( "ProdDataInterfaceHmi".cycleTimerDataSet[3].control[20].run )
   END_RUNG
   // the same network as SCL:
   "ProdDataInterfaceHmi".cycleTimerDataSet[3].control[1].run := #TRUE AND ("Unit1.Em2.HmiInterface".semiAutoSplice.jobs.status.activeJobNumber = "U1EM2_JOB01");
   "ProdDataInterfaceHmi".cycleTimerDataSet[3].control[2].run := #TRUE AND ("Unit1.Em2.HmiInterface".semiAutoSplice.jobs.status.activeJobNumber = "U1EM2_JOB02");
   "ProdDataInterfaceHmi".cycleTimerDataSet[3].control[3].run := #TRUE AND ("Unit1.Em2.HmiInterface".semiAutoSplice.jobs.status.activeJobNumber = "U1EM2_JOB03");
   "ProdDataInterfaceHmi".cycleTimerDataSet[3].control[4].run := #TRUE AND ("Unit1.Em2.HmiInterface".semiAutoSplice.jobs.status.activeJobNumber = "U1EM2_JOB04");
   "ProdDataInterfaceHmi".cycleTimerDataSet[3].control[5].run := #TRUE AND ("Unit1.Em2.HmiInterface".semiAutoSplice.jobs.status.activeJobNumber = "U1EM2_JOB05");
   "ProdDataInterfaceHmi".cycleTimerDataSet[3].control[6].run := #TRUE AND ("Unit1.Em2.HmiInterface".semiAutoSplice.jobs.status.activeJobNumber = "U1EM2_JOB06");
   "ProdDataInterfaceHmi".cycleTimerDataSet[3].control[7].run := #TRUE AND ("Unit1.Em2.HmiInterface".semiAutoSplice.jobs.status.activeJobNumber = "U1EM2_JOB07");
   "ProdDataInterfaceHmi".cycleTimerDataSet[3].control[8].run := #TRUE AND ("Unit1.Em2.HmiInterface".semiAutoSplice.jobs.status.activeJobNumber = "U1EM2_JOB08");
   "ProdDataInterfaceHmi".cycleTimerDataSet[3].control[9].run := #TRUE AND ("Unit1.Em2.HmiInterface".semiAutoSplice.jobs.status.activeJobNumber = "U1EM2_JOB09");
   "ProdDataInterfaceHmi".cycleTimerDataSet[3].control[10].run := #TRUE AND ("Unit1.Em2.HmiInterface".semiAutoSplice.jobs.status.activeJobNumber = "U1EM2_JOB10");
   "ProdDataInterfaceHmi".cycleTimerDataSet[3].control[11].run := #TRUE AND ("Unit1.Em2.HmiInterface".semiAutoSplice.jobs.status.activeJobNumber = "U1EM2_JOB11");
   "ProdDataInterfaceHmi".cycleTimerDataSet[3].control[12].run := #TRUE AND ("Unit1.Em2.HmiInterface".semiAutoSplice.jobs.status.activeJobNumber = "U1EM2_JOB12");
   "ProdDataInterfaceHmi".cycleTimerDataSet[3].control[13].run := #TRUE AND ("Unit1.Em2.HmiInterface".semiAutoSplice.jobs.status.activeJobNumber = "U1EM2_JOB13");
   "ProdDataInterfaceHmi".cycleTimerDataSet[3].control[14].run := #TRUE AND ("Unit1.Em2.HmiInterface".semiAutoSplice.jobs.status.activeJobNumber = "U1EM2_JOB14");
   "ProdDataInterfaceHmi".cycleTimerDataSet[3].control[15].run := #TRUE AND ("Unit1.Em2.HmiInterface".semiAutoSplice.jobs.status.activeJobNumber = "U1EM2_JOB15");
   "ProdDataInterfaceHmi".cycleTimerDataSet[3].control[20].run := #TRUE AND ("Unit1.Em2.HmiInterface".semiAutoSplice.jobs.status.activeJobNumber = "U1EM2_JOB20");
END_REGION

REGION Network 4: cycleTimerDataSet[4]
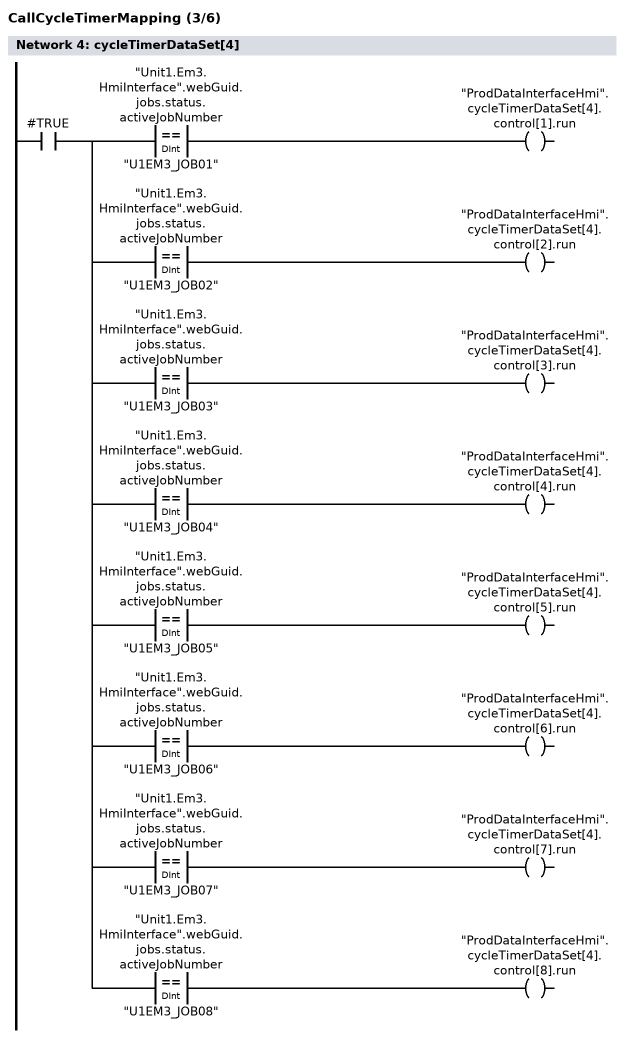
   RUNG wire#powerrail
      Contact( #TRUE )
      wire#w1
      { S7_Templates := "SrcType := DInt" } EQ_Contact(in1 := "Unit1.Em3.HmiInterface".webGuid.jobs.status.activeJobNumber, in2 := "U1EM3_JOB01")
      Coil( "ProdDataInterfaceHmi".cycleTimerDataSet[4].control[1].run )
   END_RUNG
   RUNG wire#w1
      { S7_Templates := "SrcType := DInt" } EQ_Contact(in1 := "Unit1.Em3.HmiInterface".webGuid.jobs.status.activeJobNumber, in2 := "U1EM3_JOB02")
      Coil( "ProdDataInterfaceHmi".cycleTimerDataSet[4].control[2].run )
   END_RUNG
   RUNG wire#w1
      { S7_Templates := "SrcType := DInt" } EQ_Contact(in1 := "Unit1.Em3.HmiInterface".webGuid.jobs.status.activeJobNumber, in2 := "U1EM3_JOB03")
      Coil( "ProdDataInterfaceHmi".cycleTimerDataSet[4].control[3].run )
   END_RUNG
   RUNG wire#w1
      { S7_Templates := "SrcType := DInt" } EQ_Contact(in1 := "Unit1.Em3.HmiInterface".webGuid.jobs.status.activeJobNumber, in2 := "U1EM3_JOB04")
      Coil( "ProdDataInterfaceHmi".cycleTimerDataSet[4].control[4].run )
   END_RUNG
   RUNG wire#w1
      { S7_Templates := "SrcType := DInt" } EQ_Contact(in1 := "Unit1.Em3.HmiInterface".webGuid.jobs.status.activeJobNumber, in2 := "U1EM3_JOB05")
      Coil( "ProdDataInterfaceHmi".cycleTimerDataSet[4].control[5].run )
   END_RUNG
   RUNG wire#w1
      { S7_Templates := "SrcType := DInt" } EQ_Contact(in1 := "Unit1.Em3.HmiInterface".webGuid.jobs.status.activeJobNumber, in2 := "U1EM3_JOB06")
      Coil( "ProdDataInterfaceHmi".cycleTimerDataSet[4].control[6].run )
   END_RUNG
   RUNG wire#w1
      { S7_Templates := "SrcType := DInt" } EQ_Contact(in1 := "Unit1.Em3.HmiInterface".webGuid.jobs.status.activeJobNumber, in2 := "U1EM3_JOB07")
      Coil( "ProdDataInterfaceHmi".cycleTimerDataSet[4].control[7].run )
   END_RUNG
   RUNG wire#w1
      { S7_Templates := "SrcType := DInt" } EQ_Contact(in1 := "Unit1.Em3.HmiInterface".webGuid.jobs.status.activeJobNumber, in2 := "U1EM3_JOB08")
      Coil( "ProdDataInterfaceHmi".cycleTimerDataSet[4].control[8].run )
   END_RUNG
   // the same network as SCL:
   "ProdDataInterfaceHmi".cycleTimerDataSet[4].control[1].run := #TRUE AND ("Unit1.Em3.HmiInterface".webGuid.jobs.status.activeJobNumber = "U1EM3_JOB01");
   "ProdDataInterfaceHmi".cycleTimerDataSet[4].control[2].run := #TRUE AND ("Unit1.Em3.HmiInterface".webGuid.jobs.status.activeJobNumber = "U1EM3_JOB02");
   "ProdDataInterfaceHmi".cycleTimerDataSet[4].control[3].run := #TRUE AND ("Unit1.Em3.HmiInterface".webGuid.jobs.status.activeJobNumber = "U1EM3_JOB03");
   "ProdDataInterfaceHmi".cycleTimerDataSet[4].control[4].run := #TRUE AND ("Unit1.Em3.HmiInterface".webGuid.jobs.status.activeJobNumber = "U1EM3_JOB04");
   "ProdDataInterfaceHmi".cycleTimerDataSet[4].control[5].run := #TRUE AND ("Unit1.Em3.HmiInterface".webGuid.jobs.status.activeJobNumber = "U1EM3_JOB05");
   "ProdDataInterfaceHmi".cycleTimerDataSet[4].control[6].run := #TRUE AND ("Unit1.Em3.HmiInterface".webGuid.jobs.status.activeJobNumber = "U1EM3_JOB06");
   "ProdDataInterfaceHmi".cycleTimerDataSet[4].control[7].run := #TRUE AND ("Unit1.Em3.HmiInterface".webGuid.jobs.status.activeJobNumber = "U1EM3_JOB07");
   "ProdDataInterfaceHmi".cycleTimerDataSet[4].control[8].run := #TRUE AND ("Unit1.Em3.HmiInterface".webGuid.jobs.status.activeJobNumber = "U1EM3_JOB08");
END_REGION

REGION Network 5: cycleTimerDataSet[5]
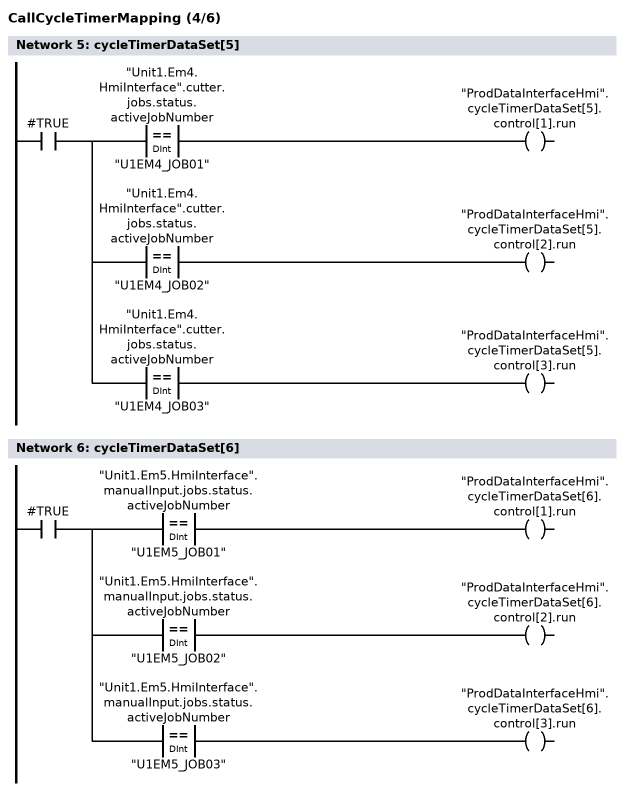
   RUNG wire#powerrail
      Contact( #TRUE )
      wire#w1
      { S7_Templates := "SrcType := DInt" } EQ_Contact(in1 := "Unit1.Em4.HmiInterface".cutter.jobs.status.activeJobNumber, in2 := "U1EM4_JOB01")
      Coil( "ProdDataInterfaceHmi".cycleTimerDataSet[5].control[1].run )
   END_RUNG
   RUNG wire#w1
      { S7_Templates := "SrcType := DInt" } EQ_Contact(in1 := "Unit1.Em4.HmiInterface".cutter.jobs.status.activeJobNumber, in2 := "U1EM4_JOB02")
      Coil( "ProdDataInterfaceHmi".cycleTimerDataSet[5].control[2].run )
   END_RUNG
   RUNG wire#w1
      { S7_Templates := "SrcType := DInt" } EQ_Contact(in1 := "Unit1.Em4.HmiInterface".cutter.jobs.status.activeJobNumber, in2 := "U1EM4_JOB03")
      Coil( "ProdDataInterfaceHmi".cycleTimerDataSet[5].control[3].run )
   END_RUNG
   // the same network as SCL:
   "ProdDataInterfaceHmi".cycleTimerDataSet[5].control[1].run := #TRUE AND ("Unit1.Em4.HmiInterface".cutter.jobs.status.activeJobNumber = "U1EM4_JOB01");
   "ProdDataInterfaceHmi".cycleTimerDataSet[5].control[2].run := #TRUE AND ("Unit1.Em4.HmiInterface".cutter.jobs.status.activeJobNumber = "U1EM4_JOB02");
   "ProdDataInterfaceHmi".cycleTimerDataSet[5].control[3].run := #TRUE AND ("Unit1.Em4.HmiInterface".cutter.jobs.status.activeJobNumber = "U1EM4_JOB03");
END_REGION

REGION Network 6: cycleTimerDataSet[6]
   RUNG wire#powerrail
      Contact( #TRUE )
      wire#w1
      { S7_Templates := "SrcType := DInt" } EQ_Contact(in1 := "Unit1.Em5.HmiInterface".manualInput.jobs.status.activeJobNumber, in2 := "U1EM5_JOB01")
      Coil( "ProdDataInterfaceHmi".cycleTimerDataSet[6].control[1].run )
   END_RUNG
   RUNG wire#w1
      { S7_Templates := "SrcType := DInt" } EQ_Contact(in1 := "Unit1.Em5.HmiInterface".manualInput.jobs.status.activeJobNumber, in2 := "U1EM5_JOB02")
      Coil( "ProdDataInterfaceHmi".cycleTimerDataSet[6].control[2].run )
   END_RUNG
   RUNG wire#w1
      { S7_Templates := "SrcType := DInt" } EQ_Contact(in1 := "Unit1.Em5.HmiInterface".manualInput.jobs.status.activeJobNumber, in2 := "U1EM5_JOB03")
      Coil( "ProdDataInterfaceHmi".cycleTimerDataSet[6].control[3].run )
   END_RUNG
   // the same network as SCL:
   "ProdDataInterfaceHmi".cycleTimerDataSet[6].control[1].run := #TRUE AND ("Unit1.Em5.HmiInterface".manualInput.jobs.status.activeJobNumber = "U1EM5_JOB01");
   "ProdDataInterfaceHmi".cycleTimerDataSet[6].control[2].run := #TRUE AND ("Unit1.Em5.HmiInterface".manualInput.jobs.status.activeJobNumber = "U1EM5_JOB02");
   "ProdDataInterfaceHmi".cycleTimerDataSet[6].control[3].run := #TRUE AND ("Unit1.Em5.HmiInterface".manualInput.jobs.status.activeJobNumber = "U1EM5_JOB03");
END_REGION

REGION Network 7: cycleTimerDataSet[7]
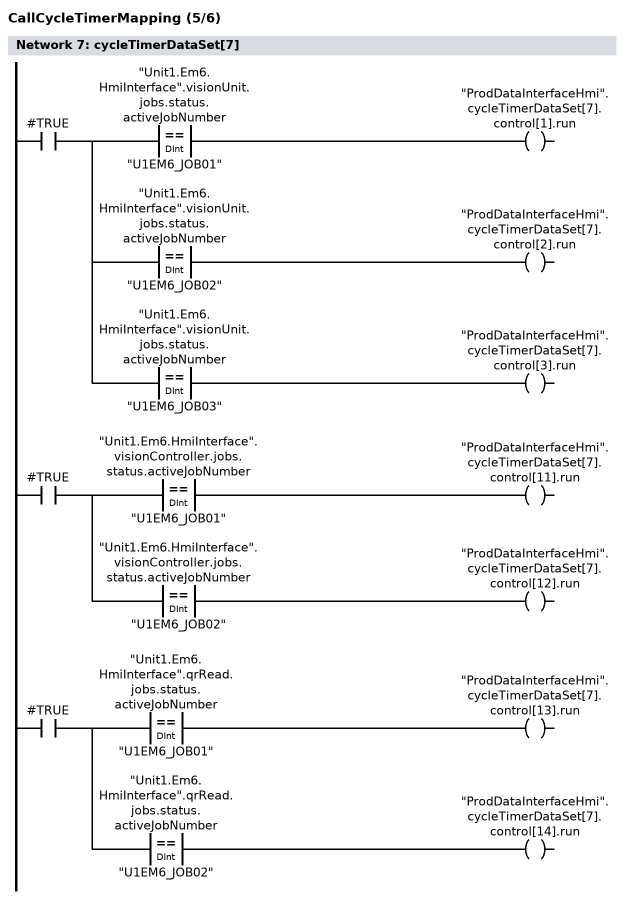
   RUNG wire#powerrail
      Contact( #TRUE )
      wire#w1
      { S7_Templates := "SrcType := DInt" } EQ_Contact(in1 := "Unit1.Em6.HmiInterface".visionUnit.jobs.status.activeJobNumber, in2 := "U1EM6_JOB01")
      Coil( "ProdDataInterfaceHmi".cycleTimerDataSet[7].control[1].run )
   END_RUNG
   RUNG wire#w1
      { S7_Templates := "SrcType := DInt" } EQ_Contact(in1 := "Unit1.Em6.HmiInterface".visionUnit.jobs.status.activeJobNumber, in2 := "U1EM6_JOB02")
      Coil( "ProdDataInterfaceHmi".cycleTimerDataSet[7].control[2].run )
   END_RUNG
   RUNG wire#w1
      { S7_Templates := "SrcType := DInt" } EQ_Contact(in1 := "Unit1.Em6.HmiInterface".visionUnit.jobs.status.activeJobNumber, in2 := "U1EM6_JOB03")
      Coil( "ProdDataInterfaceHmi".cycleTimerDataSet[7].control[3].run )
   END_RUNG
   RUNG wire#powerrail
      Contact( #TRUE )
      wire#w2
      { S7_Templates := "SrcType := DInt" } EQ_Contact(in1 := "Unit1.Em6.HmiInterface".visionController.jobs.status.activeJobNumber, in2 := "U1EM6_JOB01")
      Coil( "ProdDataInterfaceHmi".cycleTimerDataSet[7].control[11].run )
   END_RUNG
   RUNG wire#w2
      { S7_Templates := "SrcType := DInt" } EQ_Contact(in1 := "Unit1.Em6.HmiInterface".visionController.jobs.status.activeJobNumber, in2 := "U1EM6_JOB02")
      Coil( "ProdDataInterfaceHmi".cycleTimerDataSet[7].control[12].run )
   END_RUNG
   RUNG wire#powerrail
      Contact( #TRUE )
      wire#w3
      { S7_Templates := "SrcType := DInt" } EQ_Contact(in1 := "Unit1.Em6.HmiInterface".qrRead.jobs.status.activeJobNumber, in2 := "U1EM6_JOB01")
      Coil( "ProdDataInterfaceHmi".cycleTimerDataSet[7].control[13].run )
   END_RUNG
   RUNG wire#w3
      { S7_Templates := "SrcType := DInt" } EQ_Contact(in1 := "Unit1.Em6.HmiInterface".qrRead.jobs.status.activeJobNumber, in2 := "U1EM6_JOB02")
      Coil( "ProdDataInterfaceHmi".cycleTimerDataSet[7].control[14].run )
   END_RUNG
   // the same network as SCL:
   "ProdDataInterfaceHmi".cycleTimerDataSet[7].control[1].run := #TRUE AND ("Unit1.Em6.HmiInterface".visionUnit.jobs.status.activeJobNumber = "U1EM6_JOB01");
   "ProdDataInterfaceHmi".cycleTimerDataSet[7].control[2].run := #TRUE AND ("Unit1.Em6.HmiInterface".visionUnit.jobs.status.activeJobNumber = "U1EM6_JOB02");
   "ProdDataInterfaceHmi".cycleTimerDataSet[7].control[3].run := #TRUE AND ("Unit1.Em6.HmiInterface".visionUnit.jobs.status.activeJobNumber = "U1EM6_JOB03");
   "ProdDataInterfaceHmi".cycleTimerDataSet[7].control[11].run := #TRUE AND ("Unit1.Em6.HmiInterface".visionController.jobs.status.activeJobNumber = "U1EM6_JOB01");
   "ProdDataInterfaceHmi".cycleTimerDataSet[7].control[12].run := #TRUE AND ("Unit1.Em6.HmiInterface".visionController.jobs.status.activeJobNumber = "U1EM6_JOB02");
   "ProdDataInterfaceHmi".cycleTimerDataSet[7].control[13].run := #TRUE AND ("Unit1.Em6.HmiInterface".qrRead.jobs.status.activeJobNumber = "U1EM6_JOB01");
   "ProdDataInterfaceHmi".cycleTimerDataSet[7].control[14].run := #TRUE AND ("Unit1.Em6.HmiInterface".qrRead.jobs.status.activeJobNumber = "U1EM6_JOB02");
END_REGION

REGION Network 8: cycleTimerDataSet[8]
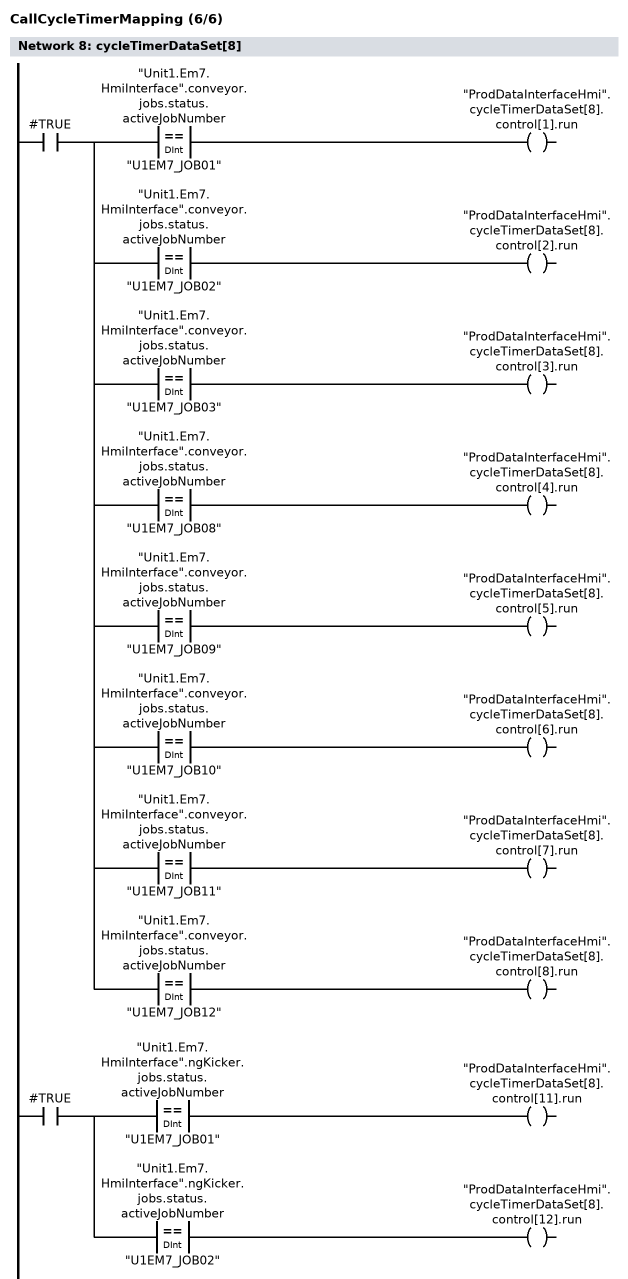
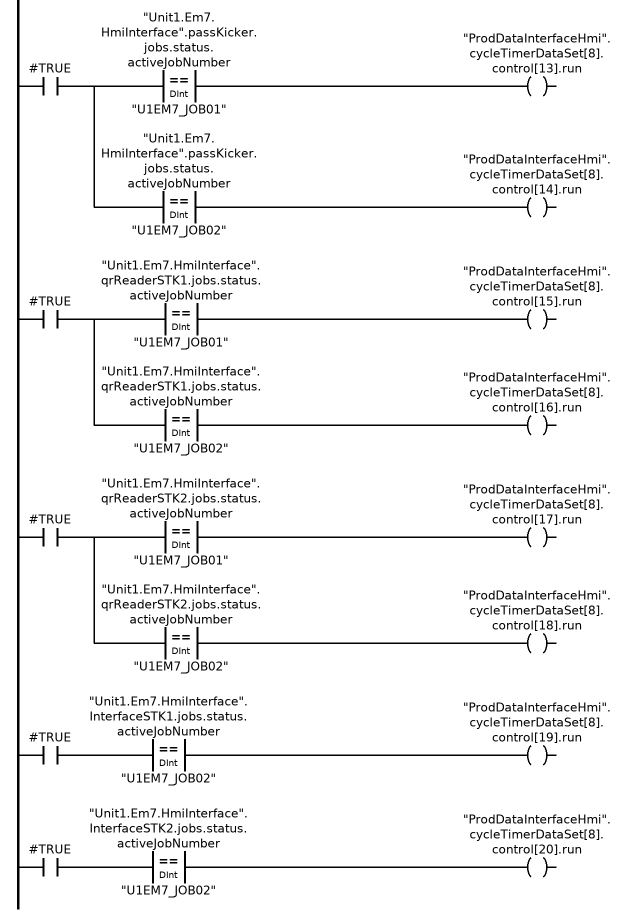
   RUNG wire#powerrail
      Contact( #TRUE )
      wire#w1
      { S7_Templates := "SrcType := DInt" } EQ_Contact(in1 := "Unit1.Em7.HmiInterface".conveyor.jobs.status.activeJobNumber, in2 := "U1EM7_JOB01")
      Coil( "ProdDataInterfaceHmi".cycleTimerDataSet[8].control[1].run )
   END_RUNG
   RUNG wire#w1
      { S7_Templates := "SrcType := DInt" } EQ_Contact(in1 := "Unit1.Em7.HmiInterface".conveyor.jobs.status.activeJobNumber, in2 := "U1EM7_JOB02")
      Coil( "ProdDataInterfaceHmi".cycleTimerDataSet[8].control[2].run )
   END_RUNG
   RUNG wire#w1
      { S7_Templates := "SrcType := DInt" } EQ_Contact(in1 := "Unit1.Em7.HmiInterface".conveyor.jobs.status.activeJobNumber, in2 := "U1EM7_JOB03")
      Coil( "ProdDataInterfaceHmi".cycleTimerDataSet[8].control[3].run )
   END_RUNG
   RUNG wire#w1
      { S7_Templates := "SrcType := DInt" } EQ_Contact(in1 := "Unit1.Em7.HmiInterface".conveyor.jobs.status.activeJobNumber, in2 := "U1EM7_JOB08")
      Coil( "ProdDataInterfaceHmi".cycleTimerDataSet[8].control[4].run )
   END_RUNG
   RUNG wire#w1
      { S7_Templates := "SrcType := DInt" } EQ_Contact(in1 := "Unit1.Em7.HmiInterface".conveyor.jobs.status.activeJobNumber, in2 := "U1EM7_JOB09")
      Coil( "ProdDataInterfaceHmi".cycleTimerDataSet[8].control[5].run )
   END_RUNG
   RUNG wire#w1
      { S7_Templates := "SrcType := DInt" } EQ_Contact(in1 := "Unit1.Em7.HmiInterface".conveyor.jobs.status.activeJobNumber, in2 := "U1EM7_JOB10")
      Coil( "ProdDataInterfaceHmi".cycleTimerDataSet[8].control[6].run )
   END_RUNG
   RUNG wire#w1
      { S7_Templates := "SrcType := DInt" } EQ_Contact(in1 := "Unit1.Em7.HmiInterface".conveyor.jobs.status.activeJobNumber, in2 := "U1EM7_JOB11")
      Coil( "ProdDataInterfaceHmi".cycleTimerDataSet[8].control[7].run )
   END_RUNG
   RUNG wire#w1
      { S7_Templates := "SrcType := DInt" } EQ_Contact(in1 := "Unit1.Em7.HmiInterface".conveyor.jobs.status.activeJobNumber, in2 := "U1EM7_JOB12")
      Coil( "ProdDataInterfaceHmi".cycleTimerDataSet[8].control[8].run )
   END_RUNG
   RUNG wire#powerrail
      Contact( #TRUE )
      wire#w2
      { S7_Templates := "SrcType := DInt" } EQ_Contact(in1 := "Unit1.Em7.HmiInterface".ngKicker.jobs.status.activeJobNumber, in2 := "U1EM7_JOB01")
      Coil( "ProdDataInterfaceHmi".cycleTimerDataSet[8].control[11].run )
   END_RUNG
   RUNG wire#w2
      { S7_Templates := "SrcType := DInt" } EQ_Contact(in1 := "Unit1.Em7.HmiInterface".ngKicker.jobs.status.activeJobNumber, in2 := "U1EM7_JOB02")
      Coil( "ProdDataInterfaceHmi".cycleTimerDataSet[8].control[12].run )
   END_RUNG
   RUNG wire#powerrail
      Contact( #TRUE )
      wire#w3
      { S7_Templates := "SrcType := DInt" } EQ_Contact(in1 := "Unit1.Em7.HmiInterface".passKicker.jobs.status.activeJobNumber, in2 := "U1EM7_JOB01")
      Coil( "ProdDataInterfaceHmi".cycleTimerDataSet[8].control[13].run )
   END_RUNG
   RUNG wire#w3
      { S7_Templates := "SrcType := DInt" } EQ_Contact(in1 := "Unit1.Em7.HmiInterface".passKicker.jobs.status.activeJobNumber, in2 := "U1EM7_JOB02")
      Coil( "ProdDataInterfaceHmi".cycleTimerDataSet[8].control[14].run )
   END_RUNG
   RUNG wire#powerrail
      Contact( #TRUE )
      wire#w4
      { S7_Templates := "SrcType := DInt" } EQ_Contact(in1 := "Unit1.Em7.HmiInterface".qrReaderSTK1.jobs.status.activeJobNumber, in2 := "U1EM7_JOB01")
      Coil( "ProdDataInterfaceHmi".cycleTimerDataSet[8].control[15].run )
   END_RUNG
   RUNG wire#w4
      { S7_Templates := "SrcType := DInt" } EQ_Contact(in1 := "Unit1.Em7.HmiInterface".qrReaderSTK1.jobs.status.activeJobNumber, in2 := "U1EM7_JOB02")
      Coil( "ProdDataInterfaceHmi".cycleTimerDataSet[8].control[16].run )
   END_RUNG
   RUNG wire#powerrail
      Contact( #TRUE )
      wire#w5
      { S7_Templates := "SrcType := DInt" } EQ_Contact(in1 := "Unit1.Em7.HmiInterface".qrReaderSTK2.jobs.status.activeJobNumber, in2 := "U1EM7_JOB01")
      Coil( "ProdDataInterfaceHmi".cycleTimerDataSet[8].control[17].run )
   END_RUNG
   RUNG wire#w5
      { S7_Templates := "SrcType := DInt" } EQ_Contact(in1 := "Unit1.Em7.HmiInterface".qrReaderSTK2.jobs.status.activeJobNumber, in2 := "U1EM7_JOB02")
      Coil( "ProdDataInterfaceHmi".cycleTimerDataSet[8].control[18].run )
   END_RUNG
   RUNG wire#powerrail
      Contact( #TRUE )
      { S7_Templates := "SrcType := DInt" } EQ_Contact(in1 := "Unit1.Em7.HmiInterface".InterfaceSTK1.jobs.status.activeJobNumber, in2 := "U1EM7_JOB02")
      Coil( "ProdDataInterfaceHmi".cycleTimerDataSet[8].control[19].run )
   END_RUNG
   RUNG wire#powerrail
      Contact( #TRUE )
      { S7_Templates := "SrcType := DInt" } EQ_Contact(in1 := "Unit1.Em7.HmiInterface".InterfaceSTK2.jobs.status.activeJobNumber, in2 := "U1EM7_JOB02")
      Coil( "ProdDataInterfaceHmi".cycleTimerDataSet[8].control[20].run )
   END_RUNG
   // the same network as SCL:
   "ProdDataInterfaceHmi".cycleTimerDataSet[8].control[1].run := #TRUE AND ("Unit1.Em7.HmiInterface".conveyor.jobs.status.activeJobNumber = "U1EM7_JOB01");
   "ProdDataInterfaceHmi".cycleTimerDataSet[8].control[2].run := #TRUE AND ("Unit1.Em7.HmiInterface".conveyor.jobs.status.activeJobNumber = "U1EM7_JOB02");
   "ProdDataInterfaceHmi".cycleTimerDataSet[8].control[3].run := #TRUE AND ("Unit1.Em7.HmiInterface".conveyor.jobs.status.activeJobNumber = "U1EM7_JOB03");
   "ProdDataInterfaceHmi".cycleTimerDataSet[8].control[4].run := #TRUE AND ("Unit1.Em7.HmiInterface".conveyor.jobs.status.activeJobNumber = "U1EM7_JOB08");
   "ProdDataInterfaceHmi".cycleTimerDataSet[8].control[5].run := #TRUE AND ("Unit1.Em7.HmiInterface".conveyor.jobs.status.activeJobNumber = "U1EM7_JOB09");
   "ProdDataInterfaceHmi".cycleTimerDataSet[8].control[6].run := #TRUE AND ("Unit1.Em7.HmiInterface".conveyor.jobs.status.activeJobNumber = "U1EM7_JOB10");
   "ProdDataInterfaceHmi".cycleTimerDataSet[8].control[7].run := #TRUE AND ("Unit1.Em7.HmiInterface".conveyor.jobs.status.activeJobNumber = "U1EM7_JOB11");
   "ProdDataInterfaceHmi".cycleTimerDataSet[8].control[8].run := #TRUE AND ("Unit1.Em7.HmiInterface".conveyor.jobs.status.activeJobNumber = "U1EM7_JOB12");
   "ProdDataInterfaceHmi".cycleTimerDataSet[8].control[11].run := #TRUE AND ("Unit1.Em7.HmiInterface".ngKicker.jobs.status.activeJobNumber = "U1EM7_JOB01");
   "ProdDataInterfaceHmi".cycleTimerDataSet[8].control[12].run := #TRUE AND ("Unit1.Em7.HmiInterface".ngKicker.jobs.status.activeJobNumber = "U1EM7_JOB02");
   "ProdDataInterfaceHmi".cycleTimerDataSet[8].control[13].run := #TRUE AND ("Unit1.Em7.HmiInterface".passKicker.jobs.status.activeJobNumber = "U1EM7_JOB01");
   "ProdDataInterfaceHmi".cycleTimerDataSet[8].control[14].run := #TRUE AND ("Unit1.Em7.HmiInterface".passKicker.jobs.status.activeJobNumber = "U1EM7_JOB02");
   "ProdDataInterfaceHmi".cycleTimerDataSet[8].control[15].run := #TRUE AND ("Unit1.Em7.HmiInterface".qrReaderSTK1.jobs.status.activeJobNumber = "U1EM7_JOB01");
   "ProdDataInterfaceHmi".cycleTimerDataSet[8].control[16].run := #TRUE AND ("Unit1.Em7.HmiInterface".qrReaderSTK1.jobs.status.activeJobNumber = "U1EM7_JOB02");
   "ProdDataInterfaceHmi".cycleTimerDataSet[8].control[17].run := #TRUE AND ("Unit1.Em7.HmiInterface".qrReaderSTK2.jobs.status.activeJobNumber = "U1EM7_JOB01");
   "ProdDataInterfaceHmi".cycleTimerDataSet[8].control[18].run := #TRUE AND ("Unit1.Em7.HmiInterface".qrReaderSTK2.jobs.status.activeJobNumber = "U1EM7_JOB02");
   "ProdDataInterfaceHmi".cycleTimerDataSet[8].control[19].run := #TRUE AND ("Unit1.Em7.HmiInterface".InterfaceSTK1.jobs.status.activeJobNumber = "U1EM7_JOB02");
   "ProdDataInterfaceHmi".cycleTimerDataSet[8].control[20].run := #TRUE AND ("Unit1.Em7.HmiInterface".InterfaceSTK2.jobs.status.activeJobNumber = "U1EM7_JOB02");
END_REGION
END_FUNCTION

FUNCTION_BLOCK "CompValEqOr"   // FB55, LAD
TITLE = COMP_VAL_==_OR_FB / COMP_VAL_==_OR
AUTHOR : SICAR
FAMILY : Miscellaneous
VERSION : 1.0
// Der Baustein vergleicht die Werte der Eingänge in1...in8 mit dem Wert des Eingangs „compareValue“ und verodert diese Vergleiche. Ist mindestens einer der Werte von in1...in8 gleich mit „compareValue“, so wird der Wert von „compareValue“ in den Output „value“ geschrieben. Andernfalls wird er mit dem Wert 0 beschrieben.  
// Anwendungsfall Beispiel: Damit kann ein "Summensignal" gebildet werden, z.B. für Produktionsdaten "Grenzwerte", womit ein Button animiert werden kann (Button "ProdData", "Grenzwerte").  
// 
// **Beispielaufruf**  
// Abbildung in Kontaktplan (KOP), ohne Parameterbeschaltung.  
// 
// **Aufrufschnittstelle**  
// Der Baustein wird im zyklischen Programm aufgerufen. In den Startup-Projekten ist der Baustein aufgerufen, für die Bildung eines Sammelsignals für die Grenzwerte der Produktionsdaten. Damit werden die Buttons  [ProdData]
// Compare the values of the inputs with the value of th input _compareValue_ generating a collective OR signal from these comparisons.
// stored: IsIECCheckEnabled true, MemoryReserve 100, SetENOAutomatically true
   VAR_INPUT
      compareValue { ExternalAccessible := 'False'; ExternalVisible := 'False'; ExternalWritable := 'False'} : UInt;   // Vergleichs Wert / Compare value
      val1 { ExternalAccessible := 'False'; ExternalVisible := 'False'; ExternalWritable := 'False'} : UInt;   // Wert 1 / value 1
      val2 { ExternalAccessible := 'False'; ExternalVisible := 'False'; ExternalWritable := 'False'} : UInt;   // Wert 2 / value 2
      val3 { ExternalAccessible := 'False'; ExternalVisible := 'False'; ExternalWritable := 'False'} : UInt;   // Wert 3 / value 3
      val4 { ExternalAccessible := 'False'; ExternalVisible := 'False'; ExternalWritable := 'False'} : UInt;   // Wert 4 / value 4
      val5 { ExternalAccessible := 'False'; ExternalVisible := 'False'; ExternalWritable := 'False'} : UInt;   // Wert 5 / value 5
      val6 { ExternalAccessible := 'False'; ExternalVisible := 'False'; ExternalWritable := 'False'} : UInt;   // Wert 6 / value 6
      val7 { ExternalAccessible := 'False'; ExternalVisible := 'False'; ExternalWritable := 'False'} : UInt;   // Wert 7 / value 7
      val8 { ExternalAccessible := 'False'; ExternalVisible := 'False'; ExternalWritable := 'False'} : UInt;   // Wert 8 / value 8
   END_VAR
   VAR_OUTPUT
      value { ExternalAccessible := 'False'; ExternalVisible := 'False'; ExternalWritable := 'False'} : UInt;   // Ergebnis Wert / Result value
   END_VAR
   VAR_TEMP
      tempDummy : Bool;   // Dummy
   END_VAR
BEGIN

REGION Network 1: Aufruf: Initialisierung SPS / ChangeLog
   // SIEMENS AG / (c)Copyright 2023
   // ------------------------------------------------------------------------------
   // Title:            CompValEqOr (FB55)
   // Comment/Function: Compare the values of the inputs with the value of th input compareValue generating a collective OR signal from these comparisons.
   // Library/Family:   Automation Framework
   // Author:           Siemens Digital Industry
   // Tested with:      ---
   // Engineering:      TIA Portal V19
   // Restrictions:     -
   // Requirements:     ---
   // ------------------------------------------------------------------------------
   // Change log table:
   // Version  | Date       | Expert in charge       | Changes applied
   // ---------|------------|------------------------|------------------------------
   // 01.00.00 | 11.12.2023 | Siemens Industry Online Support
   //                         First released version
END_REGION

REGION Network 2: Beschreibung / Description
   // The block compares the values of the inputs _in1 ... in8_ with the value of the input _compareValue_ and generates a collective OR signal from these comparisons. If at least one of the values of in1 ... in8 is equal with _compareValue_, the value of _compareValue_ is written to output “value”.  
   // Otherwise, “value” is written with the value 0.  
   // Use Case example: With this, a "summary signal" can be formed, e.g. for production data "Limit Values", with which a button can be animated (Button "ProdData", "LimitValues"). 
   // 
   // **Block call example**  
   // 
   // The call is shown as “Ladder Diagram” (LAD), without parameters.  
   // 
   // **Calling interface**  
   // 
   // The block is called in the cyclic program. In the startup projects, the block is called to generate a collective signal for the limit values of the production data. The buttons [ProdData] and [LimitValues] are animated in color, depending on the value range of the limit values.
   // 
   // **Operation mode Automatic / Manual**  
   // 
   // The block is independent of operation modes. Therefor it is not assigned to any operation mode area.
END_REGION

REGION Network 3: VALUE = 0 schreiben / set VALUE = 0
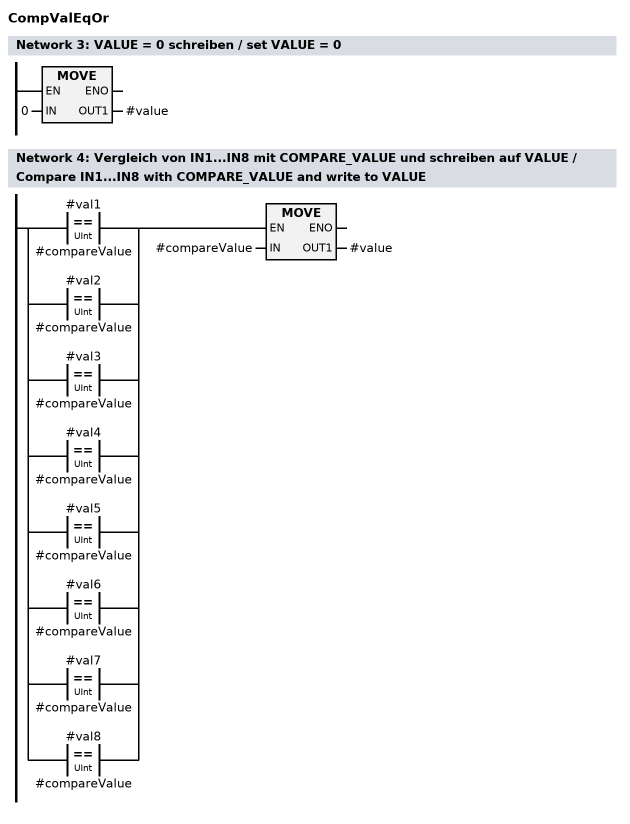
   RUNG wire#powerrail
      Move(in := 0, out1 => #value)
   END_RUNG
   // the same network as SCL:
   #value := 0;
END_REGION

REGION Network 4: Vergleich von IN1...IN8 mit COMPARE_VALUE und schreiben auf VALUE / Compare IN1...IN8 with COMPARE_VALUE and write to VALUE
   RUNG wire#powerrail
      { S7_Templates := "SrcType := UInt" } EQ_Contact(in1 := #val1, in2 := #compareValue)
      wire#w1
      Move(in := #compareValue, out1 => #value)
   END_RUNG
   RUNG wire#powerrail
      { S7_Templates := "SrcType := UInt" } EQ_Contact(in1 := #val2, in2 := #compareValue)
   END_RUNG wire#w1
   RUNG wire#powerrail
      { S7_Templates := "SrcType := UInt" } EQ_Contact(in1 := #val3, in2 := #compareValue)
   END_RUNG wire#w1
   RUNG wire#powerrail
      { S7_Templates := "SrcType := UInt" } EQ_Contact(in1 := #val4, in2 := #compareValue)
   END_RUNG wire#w1
   RUNG wire#powerrail
      { S7_Templates := "SrcType := UInt" } EQ_Contact(in1 := #val5, in2 := #compareValue)
   END_RUNG wire#w1
   RUNG wire#powerrail
      { S7_Templates := "SrcType := UInt" } EQ_Contact(in1 := #val6, in2 := #compareValue)
   END_RUNG wire#w1
   RUNG wire#powerrail
      { S7_Templates := "SrcType := UInt" } EQ_Contact(in1 := #val7, in2 := #compareValue)
   END_RUNG wire#w1
   RUNG wire#powerrail
      { S7_Templates := "SrcType := UInt" } EQ_Contact(in1 := #val8, in2 := #compareValue)
   END_RUNG wire#w1
   // the same network as SCL:
   IF (#val1 = #compareValue) OR (#val2 = #compareValue) OR (#val3 = #compareValue) OR (#val4 = #compareValue) OR (#val5 = #compareValue) OR (#val6 = #compareValue) OR (#val7 = #compareValue) OR (#val8 = #compareValue) THEN
       #value := #compareValue;
   END_IF;
END_REGION
END_FUNCTION_BLOCK

FUNCTION "CallAlarmCountMapping" : Void   // FC6, LAD
// stored: SetENOAutomatically false
BEGIN

REGION Network 1: Cutter Life Count
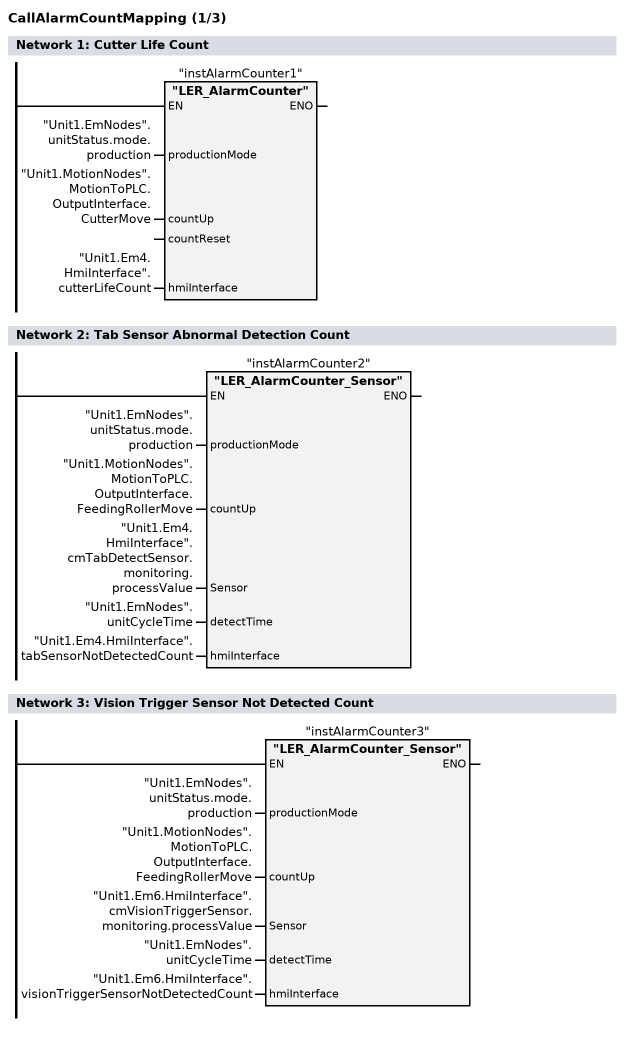
   RUNG wire#powerrail
      "instAlarmCounter1"(productionMode := "Unit1.EmNodes".unitStatus.mode.production, countUp := "Unit1.MotionNodes".MotionToPLC.OutputInterface.CutterMove, countReset :=, hmiInterface := "Unit1.Em4.HmiInterface".cutterLifeCount)
   END_RUNG
   // the same network as SCL:
   "instAlarmCounter1"(productionMode := "Unit1.EmNodes".unitStatus.mode.production,   // "LER_AlarmCounter"
                       countUp := "Unit1.MotionNodes".MotionToPLC.OutputInterface.CutterMove,
                       hmiInterface := "Unit1.Em4.HmiInterface".cutterLifeCount);
END_REGION

REGION Network 2: Tab Sensor Abnormal Detection Count
   RUNG wire#powerrail
      "instAlarmCounter2"(productionMode := "Unit1.EmNodes".unitStatus.mode.production, countUp := "Unit1.MotionNodes".MotionToPLC.OutputInterface.FeedingRollerMove, Sensor := "Unit1.Em4.HmiInterface".cmTabDetectSensor.monitoring.processValue, detectTime := "Unit1.EmNodes".unitCycleTime, hmiInterface := "Unit1.Em4.HmiInterface".tabSensorNotDetectedCount)
   END_RUNG
   // the same network as SCL:
   "instAlarmCounter2"(productionMode := "Unit1.EmNodes".unitStatus.mode.production,   // "LER_AlarmCounter_Sensor"
                       countUp := "Unit1.MotionNodes".MotionToPLC.OutputInterface.FeedingRollerMove,
                       Sensor := "Unit1.Em4.HmiInterface".cmTabDetectSensor.monitoring.processValue,
                       detectTime := "Unit1.EmNodes".unitCycleTime,
                       hmiInterface := "Unit1.Em4.HmiInterface".tabSensorNotDetectedCount);
END_REGION

REGION Network 3: Vision Trigger Sensor Not Detected Count
   RUNG wire#powerrail
      "instAlarmCounter3"(productionMode := "Unit1.EmNodes".unitStatus.mode.production, countUp := "Unit1.MotionNodes".MotionToPLC.OutputInterface.FeedingRollerMove, Sensor := "Unit1.Em6.HmiInterface".cmVisionTriggerSensor.monitoring.processValue, detectTime := "Unit1.EmNodes".unitCycleTime, hmiInterface := "Unit1.Em6.HmiInterface".visionTriggerSensorNotDetectedCount)
   END_RUNG
   // the same network as SCL:
   "instAlarmCounter3"(productionMode := "Unit1.EmNodes".unitStatus.mode.production,   // "LER_AlarmCounter_Sensor"
                       countUp := "Unit1.MotionNodes".MotionToPLC.OutputInterface.FeedingRollerMove,
                       Sensor := "Unit1.Em6.HmiInterface".cmVisionTriggerSensor.monitoring.processValue,
                       detectTime := "Unit1.EmNodes".unitCycleTime,
                       hmiInterface := "Unit1.Em6.HmiInterface".visionTriggerSensorNotDetectedCount);
END_REGION

REGION Network 4: Ng Kicker Sensor Not Detected Count
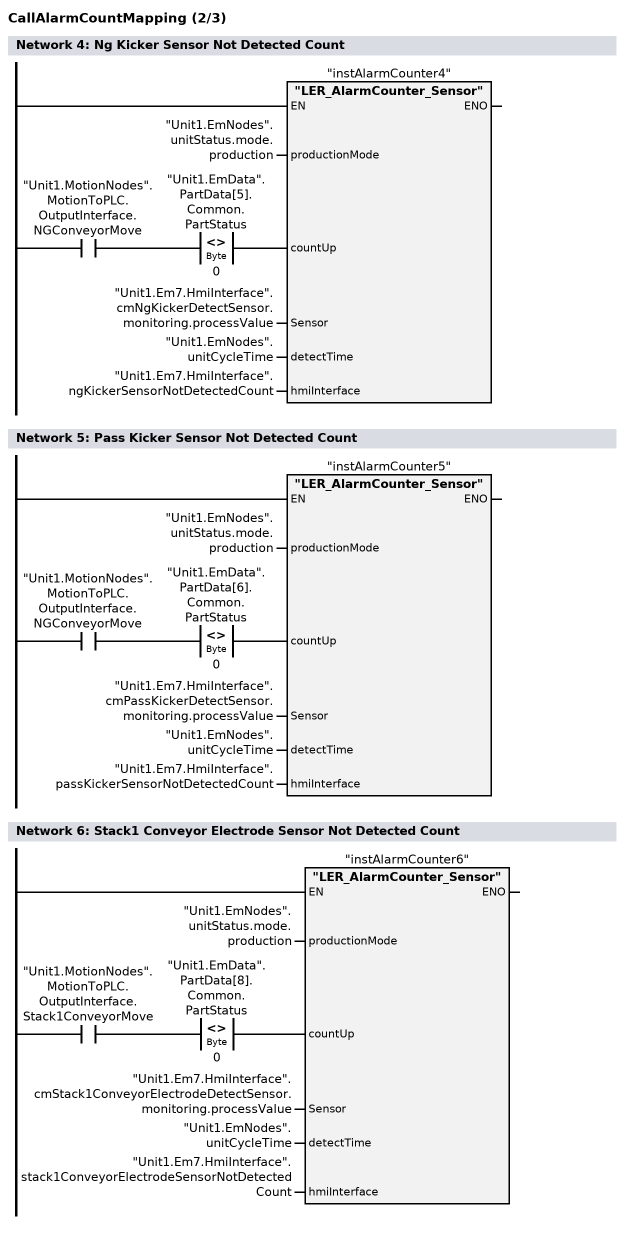
   RUNG wire#powerrail
      "instAlarmCounter4"(countUp := wire#w1, productionMode := "Unit1.EmNodes".unitStatus.mode.production, Sensor := "Unit1.Em7.HmiInterface".cmNgKickerDetectSensor.monitoring.processValue, detectTime := "Unit1.EmNodes".unitCycleTime, hmiInterface := "Unit1.Em7.HmiInterface".ngKickerSensorNotDetectedCount)
   END_RUNG
   RUNG wire#powerrail
      Contact( "Unit1.MotionNodes".MotionToPLC.OutputInterface.NGConveyorMove )
      { S7_Templates := "SrcType := Byte" } NE_Contact(in1 := "Unit1.EmData".PartData[5].Common.PartStatus, in2 := 0)
   END_RUNG wire#w1
   // the same network as SCL:
   "instAlarmCounter4"(productionMode := "Unit1.EmNodes".unitStatus.mode.production,   // "LER_AlarmCounter_Sensor"
                       countUp := "Unit1.MotionNodes".MotionToPLC.OutputInterface.NGConveyorMove AND ("Unit1.EmData".PartData[5].Common.PartStatus <> 0),
                       Sensor := "Unit1.Em7.HmiInterface".cmNgKickerDetectSensor.monitoring.processValue,
                       detectTime := "Unit1.EmNodes".unitCycleTime,
                       hmiInterface := "Unit1.Em7.HmiInterface".ngKickerSensorNotDetectedCount);
END_REGION

REGION Network 5: Pass Kicker Sensor Not Detected Count
   RUNG wire#powerrail
      "instAlarmCounter5"(countUp := wire#w1, productionMode := "Unit1.EmNodes".unitStatus.mode.production, Sensor := "Unit1.Em7.HmiInterface".cmPassKickerDetectSensor.monitoring.processValue, detectTime := "Unit1.EmNodes".unitCycleTime, hmiInterface := "Unit1.Em7.HmiInterface".passKickerSensorNotDetectedCount)
   END_RUNG
   RUNG wire#powerrail
      Contact( "Unit1.MotionNodes".MotionToPLC.OutputInterface.NGConveyorMove )
      { S7_Templates := "SrcType := Byte" } NE_Contact(in1 := "Unit1.EmData".PartData[6].Common.PartStatus, in2 := 0)
   END_RUNG wire#w1
   // the same network as SCL:
   "instAlarmCounter5"(productionMode := "Unit1.EmNodes".unitStatus.mode.production,   // "LER_AlarmCounter_Sensor"
                       countUp := "Unit1.MotionNodes".MotionToPLC.OutputInterface.NGConveyorMove AND ("Unit1.EmData".PartData[6].Common.PartStatus <> 0),
                       Sensor := "Unit1.Em7.HmiInterface".cmPassKickerDetectSensor.monitoring.processValue,
                       detectTime := "Unit1.EmNodes".unitCycleTime,
                       hmiInterface := "Unit1.Em7.HmiInterface".passKickerSensorNotDetectedCount);
END_REGION

REGION Network 6: Stack1 Conveyor Electrode Sensor Not Detected Count
   RUNG wire#powerrail
      "instAlarmCounter6"(countUp := wire#w1, productionMode := "Unit1.EmNodes".unitStatus.mode.production, Sensor := "Unit1.Em7.HmiInterface".cmStack1ConveyorElectrodeDetectSensor.monitoring.processValue, detectTime := "Unit1.EmNodes".unitCycleTime, hmiInterface := "Unit1.Em7.HmiInterface".stack1ConveyorElectrodeSensorNotDetectedCount)
   END_RUNG
   RUNG wire#powerrail
      Contact( "Unit1.MotionNodes".MotionToPLC.OutputInterface.Stack1ConveyorMove )
      { S7_Templates := "SrcType := Byte" } NE_Contact(in1 := "Unit1.EmData".PartData[8].Common.PartStatus, in2 := 0)
   END_RUNG wire#w1
   // the same network as SCL:
   "instAlarmCounter6"(productionMode := "Unit1.EmNodes".unitStatus.mode.production,   // "LER_AlarmCounter_Sensor"
                       countUp := "Unit1.MotionNodes".MotionToPLC.OutputInterface.Stack1ConveyorMove AND ("Unit1.EmData".PartData[8].Common.PartStatus <> 0),
                       Sensor := "Unit1.Em7.HmiInterface".cmStack1ConveyorElectrodeDetectSensor.monitoring.processValue,
                       detectTime := "Unit1.EmNodes".unitCycleTime,
                       hmiInterface := "Unit1.Em7.HmiInterface".stack1ConveyorElectrodeSensorNotDetectedCount);
END_REGION

REGION Network 7: Stack2 Conveyor Electrode Sensor Not Detected Count
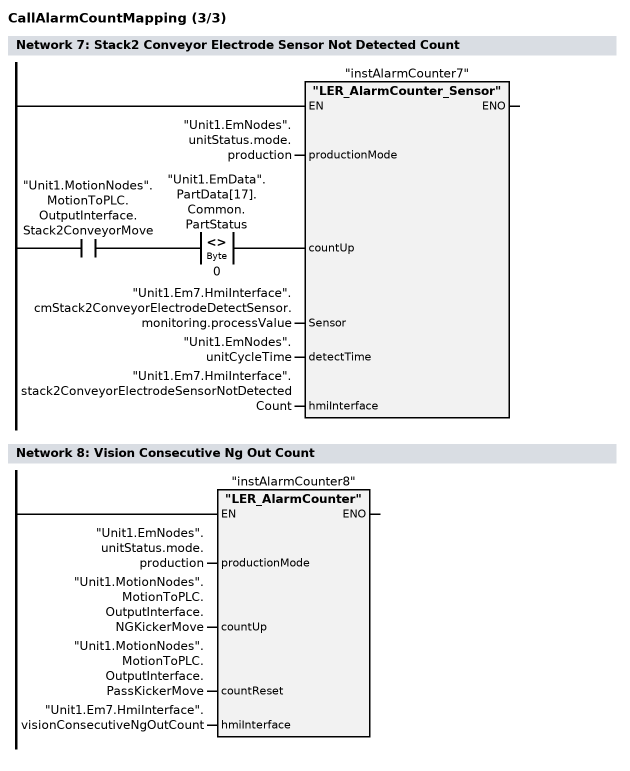
   RUNG wire#powerrail
      "instAlarmCounter7"(countUp := wire#w1, productionMode := "Unit1.EmNodes".unitStatus.mode.production, Sensor := "Unit1.Em7.HmiInterface".cmStack2ConveyorElectrodeDetectSensor.monitoring.processValue, detectTime := "Unit1.EmNodes".unitCycleTime, hmiInterface := "Unit1.Em7.HmiInterface".stack2ConveyorElectrodeSensorNotDetectedCount)
   END_RUNG
   RUNG wire#powerrail
      Contact( "Unit1.MotionNodes".MotionToPLC.OutputInterface.Stack2ConveyorMove )
      { S7_Templates := "SrcType := Byte" } NE_Contact(in1 := "Unit1.EmData".PartData[17].Common.PartStatus, in2 := 0)
   END_RUNG wire#w1
   // the same network as SCL:
   "instAlarmCounter7"(productionMode := "Unit1.EmNodes".unitStatus.mode.production,   // "LER_AlarmCounter_Sensor"
                       countUp := "Unit1.MotionNodes".MotionToPLC.OutputInterface.Stack2ConveyorMove AND ("Unit1.EmData".PartData[17].Common.PartStatus <> 0),
                       Sensor := "Unit1.Em7.HmiInterface".cmStack2ConveyorElectrodeDetectSensor.monitoring.processValue,
                       detectTime := "Unit1.EmNodes".unitCycleTime,
                       hmiInterface := "Unit1.Em7.HmiInterface".stack2ConveyorElectrodeSensorNotDetectedCount);
END_REGION

REGION Network 8: Vision Consecutive Ng Out Count
   RUNG wire#powerrail
      "instAlarmCounter8"(productionMode := "Unit1.EmNodes".unitStatus.mode.production, countUp := "Unit1.MotionNodes".MotionToPLC.OutputInterface.NGKickerMove, countReset := "Unit1.MotionNodes".MotionToPLC.OutputInterface.PassKickerMove, hmiInterface := "Unit1.Em7.HmiInterface".visionConsecutiveNgOutCount)
   END_RUNG
   // the same network as SCL:
   "instAlarmCounter8"(productionMode := "Unit1.EmNodes".unitStatus.mode.production,   // "LER_AlarmCounter"
                       countUp := "Unit1.MotionNodes".MotionToPLC.OutputInterface.NGKickerMove,
                       countReset := "Unit1.MotionNodes".MotionToPLC.OutputInterface.PassKickerMove,
                       hmiInterface := "Unit1.Em7.HmiInterface".visionConsecutiveNgOutCount);
END_REGION
END_FUNCTION

FUNCTION "CallEnergy" : Void   // FC5, LAD
TITLE = CallEnergy
// Call of Demo EnergyMeter and Energy Efficient M for EEMM demonstration
// stored: IsIECCheckEnabled true, SetENOAutomatically true
BEGIN

REGION Network 1: BLOCK INFO HEADER
   // SIEMENS AG / (c)Copyright 2023
   // ------------------------------------------------------------------------------
   // Title:            CallEnergy (FC5)
   // Comment/Function: Call of Demo EnergyMeter and Energy Efficient M for EEMM demonstration
   // Library/Family:   Energy
   // Author:           SICAR
   // Tested with:      ---
   // Engineering:      TIA Portal V19
   // Restrictions:     -
   // Requirements:     ---
   // ------------------------------------------------------------------------------
   // Change log table:
   // Version  | Date       | Expert in charge       | Changes applied
   // ---------|------------|------------------------|------------------------------
   // 01.00.00 | 11.12.2023 | SICAR
   //                         First released version
END_REGION

REGION Network 2: Call: Demo EnergyMeter, Energy Efficient M
   // Call for EEM demonstration
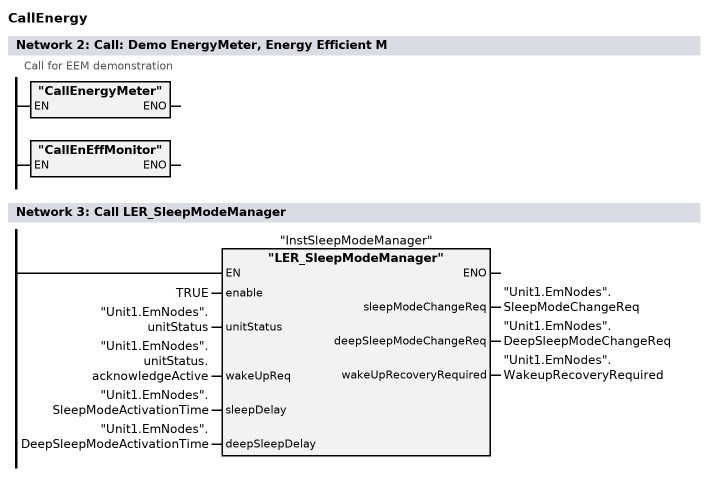
   RUNG wire#powerrail
      "CallEnergyMeter"()
   END_RUNG
   RUNG wire#powerrail
      "CallEnEffMonitor"()
   END_RUNG
   // the same network as SCL:
   "CallEnergyMeter"();
   "CallEnEffMonitor"();
END_REGION

REGION Network 3: Call LER_SleepModeManager
   RUNG wire#powerrail
      "InstSleepModeManager"(enable := TRUE, unitStatus := "Unit1.EmNodes".unitStatus, wakeUpReq := "Unit1.EmNodes".unitStatus.acknowledgeActive, sleepDelay := "Unit1.EmNodes".SleepModeActivationTime, deepSleepDelay := "Unit1.EmNodes".DeepSleepModeActivationTime, sleepModeChangeReq => "Unit1.EmNodes".SleepModeChangeReq, deepSleepModeChangeReq => "Unit1.EmNodes".DeepSleepModeChangeReq, wakeUpRecoveryRequired => "Unit1.EmNodes".WakeupRecoveryRequired)
   END_RUNG
   // the same network as SCL:
   "InstSleepModeManager"(enable := TRUE,   // "LER_SleepModeManager"
                          unitStatus := "Unit1.EmNodes".unitStatus,
                          wakeUpReq := "Unit1.EmNodes".unitStatus.acknowledgeActive,
                          sleepDelay := "Unit1.EmNodes".SleepModeActivationTime,
                          deepSleepDelay := "Unit1.EmNodes".DeepSleepModeActivationTime,
                          sleepModeChangeReq => "Unit1.EmNodes".SleepModeChangeReq,
                          deepSleepModeChangeReq => "Unit1.EmNodes".DeepSleepModeChangeReq,
                          wakeUpRecoveryRequired => "Unit1.EmNodes".WakeupRecoveryRequired);
END_REGION
END_FUNCTION

FUNCTION "CallEnergyMeter" : Void   // FC9, LAD
TITLE = CALL_AIEnergyMeter_FC
AUTHOR : SICAR
FAMILY : Energy
VERSION : 1.0
// This block calls the blocks for the AI-Energy-management.
// For more informations see SICAR userdefined documentation / SICAR online-help.
// stored: IsIECCheckEnabled true, SetENOAutomatically true
   VAR_TEMP
      tempCommResourceCounter : Int;   // für FB-Aufruf: E2M_1500_AIEnergyMeter_DRV
      tempBitsHmi : "typeEnMeterBits";   // für FB-Aufruf: E2M_1500_AIEnergyMeter_DRV
   END_VAR
   // Ret_Val : Ret_Val
BEGIN

REGION Network 1: ChangeLog
   // SIEMENS AG / (c)Copyright 2023
   // ------------------------------------------------------------------------------
   // Title:            CallEnergyMeter (FC9)
   // Comment/Function: This block calls the blocks for the AI-Energy-management.
   // Library/Family:   Automation Framework
   // Author:           Siemens Digital Industry
   // Tested with:      ---
   // Engineering:      TIA Portal V19
   // Restrictions:     -
   // Requirements:     ---
   // ------------------------------------------------------------------------------
   // Change log table:
   // Version  | Date       | Expert in charge       | Changes applied
   // ---------|------------|------------------------|------------------------------
   // 05.00.00 | 01.09.2023 | SICAR
   //                         First released version
END_REGION

REGION Network 2: AI_EnergyMeter 1
   // Call of E2MenergyMeterDrv FB
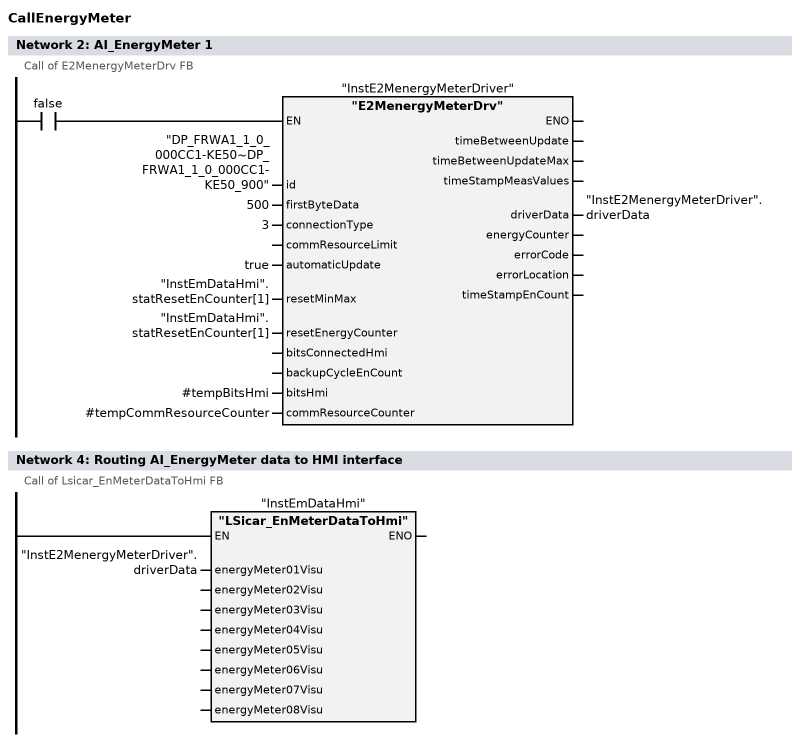
   RUNG wire#powerrail
      Contact( false )
      "InstE2MenergyMeterDriver"(id := "DP_FRWA1_1_0_000CC1-KE50~DP_FRWA1_1_0_000CC1-KE50_900", firstByteData := 500, connectionType := 3, commResourceLimit :=, automaticUpdate := true, resetMinMax := "InstEmDataHmi".statResetEnCounter[1], resetEnergyCounter := "InstEmDataHmi".statResetEnCounter[1], bitsConnectedHmi :=, backupCycleEnCount :=, bitsHmi := #tempBitsHmi, commResourceCounter := #tempCommResourceCounter, timeBetweenUpdate =>, timeBetweenUpdateMax =>, timeStampMeasValues =>, driverData => "InstE2MenergyMeterDriver".driverData, energyCounter =>, errorCode =>, errorLocation =>, timeStampEnCount =>)
   END_RUNG
   // the same network as SCL:
   IF false THEN
       "InstE2MenergyMeterDriver"(id := "DP_FRWA1_1_0_000CC1-KE50~DP_FRWA1_1_0_000CC1-KE50_900",   // "E2MenergyMeterDrv"
                               firstByteData := 500,
                               connectionType := 3,
                               automaticUpdate := true,
                               resetMinMax := "InstEmDataHmi".statResetEnCounter[1],
                               resetEnergyCounter := "InstEmDataHmi".statResetEnCounter[1],
                               bitsHmi := #tempBitsHmi,
                               commResourceCounter := #tempCommResourceCounter,
                               driverData => "InstE2MenergyMeterDriver".driverData);
   END_IF;
END_REGION

REGION Network 3 (SCL): Power meter

   // Voltage L-N
   "InstE2MenergyMeterDriver".driverData.uL1 := "PAC3220InPut"."Voltage_L1-N";
   "InstE2MenergyMeterDriver".driverData.uL2 := "PAC3220InPut"."Voltage_L2-N";
   "InstE2MenergyMeterDriver".driverData.uL3 := "PAC3220InPut"."Voltage_L3-N";
   "InstE2MenergyMeterDriver".driverData.uPhNaverage :=
   ("InstE2MenergyMeterDriver".driverData.uL1 + "InstE2MenergyMeterDriver".driverData.uL2 + "InstE2MenergyMeterDriver".driverData.uL3) / 3.0;

   IF "InstE2MenergyMeterDriver".driverData.uL1 < "InstE2MenergyMeterDriver".driverData.uL1Min OR "InstE2MenergyMeterDriver".driverData.uL1Min = 0.0 THEN
       "InstE2MenergyMeterDriver".driverData.uL1Min := "InstE2MenergyMeterDriver".driverData.uL1;
   END_IF;
   IF "InstE2MenergyMeterDriver".driverData.uL1 > "InstE2MenergyMeterDriver".driverData.uL1Max OR "InstE2MenergyMeterDriver".driverData.uL1Max = 0.0 THEN
       "InstE2MenergyMeterDriver".driverData.uL1Max := "InstE2MenergyMeterDriver".driverData.uL1;
   END_IF;

   IF "InstE2MenergyMeterDriver".driverData.uL2 < "InstE2MenergyMeterDriver".driverData.uL2Min OR "InstE2MenergyMeterDriver".driverData.uL2Min = 0.0 THEN
       "InstE2MenergyMeterDriver".driverData.uL2Min := "InstE2MenergyMeterDriver".driverData.uL2;
   END_IF;
   IF "InstE2MenergyMeterDriver".driverData.uL2 > "InstE2MenergyMeterDriver".driverData.uL2Max OR "InstE2MenergyMeterDriver".driverData.uL2Max = 0.0 THEN
       "InstE2MenergyMeterDriver".driverData.uL2Max := "InstE2MenergyMeterDriver".driverData.uL2;
   END_IF;

   IF "InstE2MenergyMeterDriver".driverData.uL3 < "InstE2MenergyMeterDriver".driverData.uL3Min OR "InstE2MenergyMeterDriver".driverData.uL3Min = 0.0 THEN
       "InstE2MenergyMeterDriver".driverData.uL3Min := "InstE2MenergyMeterDriver".driverData.uL3;
   END_IF;
   IF "InstE2MenergyMeterDriver".driverData.uL3 > "InstE2MenergyMeterDriver".driverData.uL3Max OR "InstE2MenergyMeterDriver".driverData.uL3Max = 0.0 THEN
       "InstE2MenergyMeterDriver".driverData.uL3Max := "InstE2MenergyMeterDriver".driverData.uL3;
   END_IF;

   IF "InstE2MenergyMeterDriver".driverData.uPhNaverage < "InstE2MenergyMeterDriver".driverData.uPhNaverageMin OR "InstE2MenergyMeterDriver".driverData.uPhNaverageMin = 0.0 THEN
       "InstE2MenergyMeterDriver".driverData.uPhNaverageMin := "InstE2MenergyMeterDriver".driverData.uPhNaverage;
   END_IF;
   IF "InstE2MenergyMeterDriver".driverData.uPhNaverage > "InstE2MenergyMeterDriver".driverData.uPhNaverageMax OR "InstE2MenergyMeterDriver".driverData.uPhNaverageMax = 0.0 THEN
       "InstE2MenergyMeterDriver".driverData.uPhNaverageMax := "InstE2MenergyMeterDriver".driverData.uPhNaverage;
   END_IF;

   // Voltage L-L
   "InstE2MenergyMeterDriver".driverData.uL1L2 := "PAC3220InPut"."Voltage_L1-L2";
   "InstE2MenergyMeterDriver".driverData.uL2L3 := "PAC3220InPut"."Voltage_L2-L3";
   "InstE2MenergyMeterDriver".driverData.uL3L1 := "PAC3220InPut"."Voltage_L3-L1";
   "InstE2MenergyMeterDriver".driverData.uPhPhAverage :=
   ("InstE2MenergyMeterDriver".driverData.uL1L2 + "InstE2MenergyMeterDriver".driverData.uL2L3 + "InstE2MenergyMeterDriver".driverData.uL3L1) / 3.0;

   IF "InstE2MenergyMeterDriver".driverData.uL1L2 < "InstE2MenergyMeterDriver".driverData.uL1L2Min OR "InstE2MenergyMeterDriver".driverData.uL1L2Min = 0.0 THEN
       "InstE2MenergyMeterDriver".driverData.uL1L2Min := "InstE2MenergyMeterDriver".driverData.uL1L2;
   END_IF;
   IF "InstE2MenergyMeterDriver".driverData.uL1L2 > "InstE2MenergyMeterDriver".driverData.uL1L2Max OR "InstE2MenergyMeterDriver".driverData.uL1L2Max = 0.0 THEN
       "InstE2MenergyMeterDriver".driverData.uL1L2Max := "InstE2MenergyMeterDriver".driverData.uL1L2;
   END_IF;

   IF "InstE2MenergyMeterDriver".driverData.uL2L3 < "InstE2MenergyMeterDriver".driverData.uL2L3Min OR "InstE2MenergyMeterDriver".driverData.uL2L3Min = 0.0 THEN
       "InstE2MenergyMeterDriver".driverData.uL2L3Min := "InstE2MenergyMeterDriver".driverData.uL2L3;
   END_IF;
   IF "InstE2MenergyMeterDriver".driverData.uL2L3 > "InstE2MenergyMeterDriver".driverData.uL2L3Max OR "InstE2MenergyMeterDriver".driverData.uL2L3Max = 0.0 THEN
       "InstE2MenergyMeterDriver".driverData.uL2L3Max := "InstE2MenergyMeterDriver".driverData.uL2L3;
   END_IF;

   IF "InstE2MenergyMeterDriver".driverData.uL3L1 < "InstE2MenergyMeterDriver".driverData.uL3L1Min OR "InstE2MenergyMeterDriver".driverData.uL3L1Min = 0.0 THEN
       "InstE2MenergyMeterDriver".driverData.uL3L1Min := "InstE2MenergyMeterDriver".driverData.uL3L1;
   END_IF;
   IF "InstE2MenergyMeterDriver".driverData.uL3L1 > "InstE2MenergyMeterDriver".driverData.uL3L1Max OR "InstE2MenergyMeterDriver".driverData.uL3L1Max = 0.0 THEN
       "InstE2MenergyMeterDriver".driverData.uL3L1Max := "InstE2MenergyMeterDriver".driverData.uL3L1;
   END_IF;

   IF "InstE2MenergyMeterDriver".driverData.uPhPhAverage < "InstE2MenergyMeterDriver".driverData.uPhPhAverageMin OR "InstE2MenergyMeterDriver".driverData.uPhPhAverageMin = 0.0 THEN
       "InstE2MenergyMeterDriver".driverData.uPhPhAverageMin := "InstE2MenergyMeterDriver".driverData.uPhPhAverage;
   END_IF;
   IF "InstE2MenergyMeterDriver".driverData.uPhPhAverage > "InstE2MenergyMeterDriver".driverData.uPhPhAverageMax OR "InstE2MenergyMeterDriver".driverData.uPhPhAverageMax = 0.0THEN
       "InstE2MenergyMeterDriver".driverData.uPhPhAverageMax := "InstE2MenergyMeterDriver".driverData.uPhPhAverage;
   END_IF;

   // Current
   "InstE2MenergyMeterDriver".driverData.iL1 := "PAC3220InPut".Current_L1;
   "InstE2MenergyMeterDriver".driverData.iL2 := "PAC3220InPut".Current_L2;
   "InstE2MenergyMeterDriver".driverData.iL3 := "PAC3220InPut".Current_L3;
   "InstE2MenergyMeterDriver".driverData.iAverage := "PAC3220InPut"."3-phase_average_current";

   IF "InstE2MenergyMeterDriver".driverData.iL1 < "InstE2MenergyMeterDriver".driverData.iL1Min OR "InstE2MenergyMeterDriver".driverData.iL1Min = 0.0 THEN
       "InstE2MenergyMeterDriver".driverData.iL1Min := "InstE2MenergyMeterDriver".driverData.iL1;
   END_IF;
   IF "InstE2MenergyMeterDriver".driverData.iL1 > "InstE2MenergyMeterDriver".driverData.iL1Max OR "InstE2MenergyMeterDriver".driverData.iL1Max = 0.0 THEN
       "InstE2MenergyMeterDriver".driverData.iL1Max := "InstE2MenergyMeterDriver".driverData.iL1;
   END_IF;

   IF "InstE2MenergyMeterDriver".driverData.iL2 < "InstE2MenergyMeterDriver".driverData.iL2Min OR "InstE2MenergyMeterDriver".driverData.iL2Min = 0.0 THEN
       "InstE2MenergyMeterDriver".driverData.iL2Min := "InstE2MenergyMeterDriver".driverData.iL2;
   END_IF;
   IF "InstE2MenergyMeterDriver".driverData.iL2 > "InstE2MenergyMeterDriver".driverData.iL2Max OR "InstE2MenergyMeterDriver".driverData.iL2Max = 0.0 THEN
       "InstE2MenergyMeterDriver".driverData.iL2Max := "InstE2MenergyMeterDriver".driverData.iL2;
   END_IF;

   IF "InstE2MenergyMeterDriver".driverData.iL3 < "InstE2MenergyMeterDriver".driverData.iL3Min OR "InstE2MenergyMeterDriver".driverData.iL3Min = 0.0 THEN
       "InstE2MenergyMeterDriver".driverData.iL3Min := "InstE2MenergyMeterDriver".driverData.iL3;
   END_IF;
   IF "InstE2MenergyMeterDriver".driverData.iL3 > "InstE2MenergyMeterDriver".driverData.iL3Max OR "InstE2MenergyMeterDriver".driverData.iL3Max = 0.0 THEN
       "InstE2MenergyMeterDriver".driverData.iL3Max := "InstE2MenergyMeterDriver".driverData.iL3;
   END_IF;

   IF "InstE2MenergyMeterDriver".driverData.iAverage < "InstE2MenergyMeterDriver".driverData.iAverageMin OR "InstE2MenergyMeterDriver".driverData.iAverageMin = 0.0 THEN
       "InstE2MenergyMeterDriver".driverData.iAverageMin := "InstE2MenergyMeterDriver".driverData.iAverage;
   END_IF;
   IF "InstE2MenergyMeterDriver".driverData.iAverage > "InstE2MenergyMeterDriver".driverData.iAverageMax OR "InstE2MenergyMeterDriver".driverData.iAverageMax = 0.0THEN
       "InstE2MenergyMeterDriver".driverData.iAverageMax := "InstE2MenergyMeterDriver".driverData.iAverage;
   END_IF;

   // Power factor
   "InstE2MenergyMeterDriver".driverData.cosL1 := "PAC3220InPut".Power_factor_L1;
   "InstE2MenergyMeterDriver".driverData.cosL2 := "PAC3220InPut".Power_factor_L2;
   "InstE2MenergyMeterDriver".driverData.cosL3 := "PAC3220InPut".Power_factor_L3;
   "InstE2MenergyMeterDriver".driverData.cosAverage := "PAC3220InPut".Total_power_factor;

   IF "InstE2MenergyMeterDriver".driverData.cosL1 < "InstE2MenergyMeterDriver".driverData.cosL1Min OR "InstE2MenergyMeterDriver".driverData.cosL1Min = 0.0 THEN
       "InstE2MenergyMeterDriver".driverData.cosL1Min := "InstE2MenergyMeterDriver".driverData.cosL1;
   END_IF;
   IF "InstE2MenergyMeterDriver".driverData.cosL1 > "InstE2MenergyMeterDriver".driverData.cosL1Max THEN
       "InstE2MenergyMeterDriver".driverData.cosL1Max := "InstE2MenergyMeterDriver".driverData.cosL1;
   END_IF;

   IF "InstE2MenergyMeterDriver".driverData.cosL2 < "InstE2MenergyMeterDriver".driverData.cosL2Min OR "InstE2MenergyMeterDriver".driverData.cosL2Min = 0.0 THEN
       "InstE2MenergyMeterDriver".driverData.cosL2Min := "InstE2MenergyMeterDriver".driverData.cosL2;
   END_IF;
   IF "InstE2MenergyMeterDriver".driverData.cosL2 > "InstE2MenergyMeterDriver".driverData.cosL2Max OR "InstE2MenergyMeterDriver".driverData.cosL2Max = 0.0 THEN
       "InstE2MenergyMeterDriver".driverData.cosL2Max := "InstE2MenergyMeterDriver".driverData.cosL2;
   END_IF;

   IF "InstE2MenergyMeterDriver".driverData.cosL3 < "InstE2MenergyMeterDriver".driverData.cosL3Min OR "InstE2MenergyMeterDriver".driverData.cosL3Min = 0.0 THEN
       "InstE2MenergyMeterDriver".driverData.cosL3Min := "InstE2MenergyMeterDriver".driverData.cosL3;
   END_IF;
   IF "InstE2MenergyMeterDriver".driverData.cosL3 > "InstE2MenergyMeterDriver".driverData.cosL3Max OR "InstE2MenergyMeterDriver".driverData.cosL3Max = 0.0THEN
       "InstE2MenergyMeterDriver".driverData.cosL3Max := "InstE2MenergyMeterDriver".driverData.cosL3;
   END_IF;

   IF "InstE2MenergyMeterDriver".driverData.cosAverage < "InstE2MenergyMeterDriver".driverData.cosAverageMin OR "InstE2MenergyMeterDriver".driverData.cosAverageMin = 0.0 THEN
       "InstE2MenergyMeterDriver".driverData.cosAverageMin := "InstE2MenergyMeterDriver".driverData.cosAverage;
   END_IF;
   IF "InstE2MenergyMeterDriver".driverData.cosAverage > "InstE2MenergyMeterDriver".driverData.cosAverageMax OR "InstE2MenergyMeterDriver".driverData.cosAverageMax = 0.0 THEN
       "InstE2MenergyMeterDriver".driverData.cosAverageMax := "InstE2MenergyMeterDriver".driverData.cosAverage;
   END_IF;

   // Frequency
   "InstE2MenergyMeterDriver".driverData.f := "PAC3220InPut".Line_frequency;

   IF "InstE2MenergyMeterDriver".driverData.f < "InstE2MenergyMeterDriver".driverData.fMin OR "InstE2MenergyMeterDriver".driverData.fMin = 0.0 THEN
       "InstE2MenergyMeterDriver".driverData.fMin := "InstE2MenergyMeterDriver".driverData.f;
   END_IF;
   IF "InstE2MenergyMeterDriver".driverData.f > "InstE2MenergyMeterDriver".driverData.fMax OR "InstE2MenergyMeterDriver".driverData.fMax = 0.0 THEN
       "InstE2MenergyMeterDriver".driverData.fMax := "InstE2MenergyMeterDriver".driverData.f;
   END_IF;


   // Apparent power
   "InstE2MenergyMeterDriver".driverData.sL1 := "Apparent power L1";
   "InstE2MenergyMeterDriver".driverData.sL2 := "Apparent power L2";
   "InstE2MenergyMeterDriver".driverData.sL3 := "Apparent power L3";
   "InstE2MenergyMeterDriver".driverData.sTotal := "PAC3220InPut".Total_apparent_power;

   IF "InstE2MenergyMeterDriver".driverData.sL1 < "InstE2MenergyMeterDriver".driverData.sL1Min OR "InstE2MenergyMeterDriver".driverData.sL1Min = 0.0 THEN
       "InstE2MenergyMeterDriver".driverData.sL1Min := "InstE2MenergyMeterDriver".driverData.sL1;
   END_IF;
   IF "InstE2MenergyMeterDriver".driverData.sL1 > "InstE2MenergyMeterDriver".driverData.sL1Max OR "InstE2MenergyMeterDriver".driverData.sL1Max = 0.0 THEN
       "InstE2MenergyMeterDriver".driverData.sL1Max := "InstE2MenergyMeterDriver".driverData.sL1;
   END_IF;

   IF "InstE2MenergyMeterDriver".driverData.sL2 < "InstE2MenergyMeterDriver".driverData.sL2Min OR "InstE2MenergyMeterDriver".driverData.sL2Min = 0.0 THEN
       "InstE2MenergyMeterDriver".driverData.sL2Min := "InstE2MenergyMeterDriver".driverData.sL2;
   END_IF;
   IF "InstE2MenergyMeterDriver".driverData.sL2 > "InstE2MenergyMeterDriver".driverData.sL2Max OR "InstE2MenergyMeterDriver".driverData.sL2Max = 0.0 THEN
       "InstE2MenergyMeterDriver".driverData.sL2Max := "InstE2MenergyMeterDriver".driverData.sL2;
   END_IF;

   IF "InstE2MenergyMeterDriver".driverData.sL3 < "InstE2MenergyMeterDriver".driverData.sL3Min OR "InstE2MenergyMeterDriver".driverData.sL3Min = 0.0 THEN
       "InstE2MenergyMeterDriver".driverData.sL3Min := "InstE2MenergyMeterDriver".driverData.sL3;
   END_IF;
   IF "InstE2MenergyMeterDriver".driverData.sL3 > "InstE2MenergyMeterDriver".driverData.sL3Max OR "InstE2MenergyMeterDriver".driverData.sL3Max = 0.0 THEN
       "InstE2MenergyMeterDriver".driverData.sL3Max := "InstE2MenergyMeterDriver".driverData.sL3;
   END_IF;

   IF "InstE2MenergyMeterDriver".driverData.sTotal < "InstE2MenergyMeterDriver".driverData.sTotalMin OR "InstE2MenergyMeterDriver".driverData.sTotalMin = 0.0 THEN
       "InstE2MenergyMeterDriver".driverData.sTotalMin := "InstE2MenergyMeterDriver".driverData.sTotal;
   END_IF;
   IF "InstE2MenergyMeterDriver".driverData.sTotal > "InstE2MenergyMeterDriver".driverData.sTotalMax OR "InstE2MenergyMeterDriver".driverData.sTotalMax = 0.0 THEN
       "InstE2MenergyMeterDriver".driverData.sTotalMax := "InstE2MenergyMeterDriver".driverData.sTotal;
   END_IF;

   // Active power
   "InstE2MenergyMeterDriver".driverData.pL1 := "Active power L1";
   "InstE2MenergyMeterDriver".driverData.pL2 := "Active power L2";
   "InstE2MenergyMeterDriver".driverData.pL3 := "Active power L3";
   "InstE2MenergyMeterDriver".driverData.pTotal := "PAC3220InPut".Total_active_power;

   IF "InstE2MenergyMeterDriver".driverData.pL1 < "InstE2MenergyMeterDriver".driverData.pL1Min OR "InstE2MenergyMeterDriver".driverData.pL1Min = 0.0 THEN
       "InstE2MenergyMeterDriver".driverData.pL1Min := "InstE2MenergyMeterDriver".driverData.pL1;
   END_IF;
   IF "InstE2MenergyMeterDriver".driverData.pL1 > "InstE2MenergyMeterDriver".driverData.pL1Max OR "InstE2MenergyMeterDriver".driverData.pL1Max = 0.0 THEN
       "InstE2MenergyMeterDriver".driverData.pL1Max := "InstE2MenergyMeterDriver".driverData.pL1;
   END_IF;

   IF "InstE2MenergyMeterDriver".driverData.pL2 < "InstE2MenergyMeterDriver".driverData.pL2Min OR "InstE2MenergyMeterDriver".driverData.pL2Min = 0.0 THEN
       "InstE2MenergyMeterDriver".driverData.pL2Min := "InstE2MenergyMeterDriver".driverData.pL2;
   END_IF;
   IF "InstE2MenergyMeterDriver".driverData.pL2 > "InstE2MenergyMeterDriver".driverData.pL2Max OR "InstE2MenergyMeterDriver".driverData.pL2Max = 0.0 THEN
       "InstE2MenergyMeterDriver".driverData.pL2Max := "InstE2MenergyMeterDriver".driverData.pL2;
   END_IF;

   IF "InstE2MenergyMeterDriver".driverData.pL3 < "InstE2MenergyMeterDriver".driverData.pL3Min OR "InstE2MenergyMeterDriver".driverData.pL3Min = 0.0 THEN
       "InstE2MenergyMeterDriver".driverData.pL3Min := "InstE2MenergyMeterDriver".driverData.pL3;
   END_IF;
   IF "InstE2MenergyMeterDriver".driverData.pL3 > "InstE2MenergyMeterDriver".driverData.pL3Max OR "InstE2MenergyMeterDriver".driverData.pL3Max = 0.0 THEN
       "InstE2MenergyMeterDriver".driverData.pL3Max := "InstE2MenergyMeterDriver".driverData.pL3;
   END_IF;

   IF "InstE2MenergyMeterDriver".driverData.pTotal < "InstE2MenergyMeterDriver".driverData.pTotalMin OR "InstE2MenergyMeterDriver".driverData.pTotalMin = 0.0 THEN
       "InstE2MenergyMeterDriver".driverData.pTotalMin := "InstE2MenergyMeterDriver".driverData.pTotal;
   END_IF;
   IF "InstE2MenergyMeterDriver".driverData.pTotal > "InstE2MenergyMeterDriver".driverData.pTotalMax OR "InstE2MenergyMeterDriver".driverData.pTotalMax = 0.0 THEN
       "InstE2MenergyMeterDriver".driverData.pTotalMax := "InstE2MenergyMeterDriver".driverData.pTotal;
   END_IF;

   // Reactive power
   "InstE2MenergyMeterDriver".driverData.qL1 := "Reactive power L1";
   "InstE2MenergyMeterDriver".driverData.qL2 := "Reactive power L2";
   "InstE2MenergyMeterDriver".driverData.qL3 := "Reactive power L3";
   "InstE2MenergyMeterDriver".driverData.qTotal := "PAC3220InPut"."Total_reactive_power_(VARn)";

   IF "InstE2MenergyMeterDriver".driverData.qL1 < "InstE2MenergyMeterDriver".driverData.qL1Min OR "InstE2MenergyMeterDriver".driverData.qL1Min = 0.0 THEN
       "InstE2MenergyMeterDriver".driverData.qL1Min := "InstE2MenergyMeterDriver".driverData.qL1;
   END_IF;
   IF "InstE2MenergyMeterDriver".driverData.qL1 > "InstE2MenergyMeterDriver".driverData.qL1Max OR "InstE2MenergyMeterDriver".driverData.qL1Max = 0.0 THEN
       "InstE2MenergyMeterDriver".driverData.qL1Max := "InstE2MenergyMeterDriver".driverData.qL1;
   END_IF;

   IF "InstE2MenergyMeterDriver".driverData.qL2 < "InstE2MenergyMeterDriver".driverData.qL2Min OR "InstE2MenergyMeterDriver".driverData.qL2Min = 0.0 THEN
       "InstE2MenergyMeterDriver".driverData.qL2Min := "InstE2MenergyMeterDriver".driverData.qL2;
   END_IF;
   IF "InstE2MenergyMeterDriver".driverData.qL2 > "InstE2MenergyMeterDriver".driverData.qL2Max OR "InstE2MenergyMeterDriver".driverData.qL2Max = 0.0 THEN
       "InstE2MenergyMeterDriver".driverData.qL2Max := "InstE2MenergyMeterDriver".driverData.qL2;
   END_IF;

   IF "InstE2MenergyMeterDriver".driverData.qL3 < "InstE2MenergyMeterDriver".driverData.qL3Min OR "InstE2MenergyMeterDriver".driverData.qL3Min = 0.0 THEN
       "InstE2MenergyMeterDriver".driverData.qL3Min := "InstE2MenergyMeterDriver".driverData.qL3;
   END_IF;
   IF "InstE2MenergyMeterDriver".driverData.qL3 > "InstE2MenergyMeterDriver".driverData.qL3Max OR "InstE2MenergyMeterDriver".driverData.qL3Max = 0.0 THEN
       "InstE2MenergyMeterDriver".driverData.qL3Max := "InstE2MenergyMeterDriver".driverData.qL3;
   END_IF;

   IF "InstE2MenergyMeterDriver".driverData.qTotal < "InstE2MenergyMeterDriver".driverData.qTotalMin OR "InstE2MenergyMeterDriver".driverData.qTotalMin = 0.0 THEN
       "InstE2MenergyMeterDriver".driverData.qTotalMin := "InstE2MenergyMeterDriver".driverData.qTotal;
   END_IF;
   IF "InstE2MenergyMeterDriver".driverData.qTotal > "InstE2MenergyMeterDriver".driverData.qTotalMax OR "InstE2MenergyMeterDriver".driverData.qTotalMax = 0.0 THEN
       "InstE2MenergyMeterDriver".driverData.qTotalMax := "InstE2MenergyMeterDriver".driverData.qTotal;
   END_IF;

   // Energy Tarif
   "InstE2MenergyMeterDriver".driverData.eActiveRate1Import := "Active energy import tariff 1(F)";
   "InstE2MenergyMeterDriver".driverData.eReactiveRate1Import := "Reactive energy import tariff 1 (F)";
   "InstE2MenergyMeterDriver".driverData.eApparentRate1Import := "Apparent energy tariff 1 (F)";
   "InstE2MenergyMeterDriver".driverData.eActiveRate1Export := "Active energy export tariff 1(F)";
   "InstE2MenergyMeterDriver".driverData.eReactiveRate1Export := "Reactive energy export tariff 1 (F)";






   // Reset 
   IF "InstEmDataHmi".statResetMinMaxAll  THEN

       // 모든 Min/Max 초기화 (Actual 값으로)
       "InstE2MenergyMeterDriver".driverData.uL1Min := 0.0;
       "InstE2MenergyMeterDriver".driverData.uL1Max := 0.0;
       "InstE2MenergyMeterDriver".driverData.uL2Min := 0.0;
       "InstE2MenergyMeterDriver".driverData.uL2Max := 0.0;
       "InstE2MenergyMeterDriver".driverData.uL3Min := 0.0;
       "InstE2MenergyMeterDriver".driverData.uL3Max := 0.0;

       "InstE2MenergyMeterDriver".driverData.uL1L2Min := 0.0;
       "InstE2MenergyMeterDriver".driverData.uL1L2Max := 0.0;
       "InstE2MenergyMeterDriver".driverData.uL2L3Min := 0.0;
       "InstE2MenergyMeterDriver".driverData.uL2L3Max := 0.0;
       "InstE2MenergyMeterDriver".driverData.uL3L1Min := 0.0;
       "InstE2MenergyMeterDriver".driverData.uL3L1Max := 0.0;

       "InstE2MenergyMeterDriver".driverData.uPhNaverageMin := 0.0;
       "InstE2MenergyMeterDriver".driverData.uPhNaverageMax := 0.0;

       "InstE2MenergyMeterDriver".driverData.uPhPhAverageMin := 0.0;
       "InstE2MenergyMeterDriver".driverData.uPhPhAverageMax := 0.0;

       "InstE2MenergyMeterDriver".driverData.iL1Min := 0.0;
       "InstE2MenergyMeterDriver".driverData.iL1Max := 0.0;
       "InstE2MenergyMeterDriver".driverData.iL2Min := 0.0;
       "InstE2MenergyMeterDriver".driverData.iL2Max := 0.0;
       "InstE2MenergyMeterDriver".driverData.iL3Min := 0.0;
       "InstE2MenergyMeterDriver".driverData.iL3Max := 0.0;

       "InstE2MenergyMeterDriver".driverData.iAverageMin := 0.0;
       "InstE2MenergyMeterDriver".driverData.iAverageMax := 0.0;

       "InstE2MenergyMeterDriver".driverData.cosL1Min := 0.0;
       "InstE2MenergyMeterDriver".driverData.cosL1Max := 0.0;
       "InstE2MenergyMeterDriver".driverData.cosL2Min := 0.0;
       "InstE2MenergyMeterDriver".driverData.cosL2Max := 0.0;
       "InstE2MenergyMeterDriver".driverData.cosL3Min := 0.0;
       "InstE2MenergyMeterDriver".driverData.cosL3Max := 0.0;

       "InstE2MenergyMeterDriver".driverData.cosAverageMin := 0.0;
       "InstE2MenergyMeterDriver".driverData.cosAverageMax := 0.0;

       "InstE2MenergyMeterDriver".driverData.fMin := 0.0;
       "InstE2MenergyMeterDriver".driverData.fMax := 0.0;

       "InstE2MenergyMeterDriver".driverData.pTotalMin := 0.0;
       "InstE2MenergyMeterDriver".driverData.pTotalMax := 0.0;
       "InstE2MenergyMeterDriver".driverData.qTotalMin := 0.0;
       "InstE2MenergyMeterDriver".driverData.qTotalMax := 0.0;
       "InstE2MenergyMeterDriver".driverData.sTotalMin := 0.0;
       "InstE2MenergyMeterDriver".driverData.sTotalMax := 0.0;

       "InstE2MenergyMeterDriver".driverData.sL1Min := 0.0;
       "InstE2MenergyMeterDriver".driverData.sL1Max := 0.0;
       "InstE2MenergyMeterDriver".driverData.sL2Min := 0.0;
       "InstE2MenergyMeterDriver".driverData.sL2Max := 0.0;
       "InstE2MenergyMeterDriver".driverData.sL3Min := 0.0;
       "InstE2MenergyMeterDriver".driverData.sL3Max := 0.0;

       "InstE2MenergyMeterDriver".driverData.pL1Min := 0.0;
       "InstE2MenergyMeterDriver".driverData.pL1Max := 0.0;
       "InstE2MenergyMeterDriver".driverData.pL2Min := 0.0;
       "InstE2MenergyMeterDriver".driverData.pL2Max := 0.0;
       "InstE2MenergyMeterDriver".driverData.pL3Min := 0.0;
       "InstE2MenergyMeterDriver".driverData.pL3Max := 0.0;

       "InstE2MenergyMeterDriver".driverData.qL1Min := 0.0;
       "InstE2MenergyMeterDriver".driverData.qL1Max := 0.0;
       "InstE2MenergyMeterDriver".driverData.qL2Min := 0.0;
       "InstE2MenergyMeterDriver".driverData.qL2Max := 0.0;
       "InstE2MenergyMeterDriver".driverData.qL3Min := 0.0;
       "InstE2MenergyMeterDriver".driverData.qL3Max := 0.0;

   END_IF;
END_REGION

REGION Network 4: Routing AI_EnergyMeter data to HMI interface
   // Call of Lsicar_EnMeterDataToHmi FB
   RUNG wire#powerrail
      "InstEmDataHmi"(energyMeter01Visu := "InstE2MenergyMeterDriver".driverData, energyMeter02Visu :=, energyMeter03Visu :=, energyMeter04Visu :=, energyMeter05Visu :=, energyMeter06Visu :=, energyMeter07Visu :=, energyMeter08Visu :=)
   END_RUNG
   // the same network as SCL:
   "InstEmDataHmi"(energyMeter01Visu := "InstE2MenergyMeterDriver".driverData);   // "LSicar_EnMeterDataToHmi"
END_REGION
END_FUNCTION

FUNCTION "CallEnEffMonitor" : Void   // FC32, LAD
TITLE = CallEnergyEfficencyMonitor
AUTHOR : SICAR
FAMILY : Energy_EEM
VERSION : 1.0
// EEM  Verwaltung / The S7 Energy Efficiency-Monitor (or S7 EE-Monitor) allows you to record the energy consumption of your machine in a SIMATIC controller, and to analyze the results on the basis of the energy and media requirements.
// stored: IsIECCheckEnabled true, SetENOAutomatically true
   VAR_TEMP
      tempMeasPointIndex : USInt;   // HMI Index / HMI index
      tempCycleCounterAvgCalc : DInt;   // Umrechnung zu TOD / Calculation to TOD
      tempPlantInProduction : Bool;   // Anlage produziert / Plant in production
      tempReturnValue : Int;   // Temporary value for storing the EnPi reset time / Temporärer Wert zur Speicherung der EnPi-Resetzeit
   END_VAR
   // Ret_Val : Ret_Val
   VAR_TEMP   // added for the SCL form of the ladder/FBD networks
      _w1 : Bool;
      _w2 : Bool;
      _w3 : Bool;
      _w4 : Bool;
   END_VAR
BEGIN

REGION Network 1: Änderungshistorie / BLOCK INFO HEADER
   // Die Änderungshistorie wird nur in englischer Editiersprache geführt.
   // SIEMENS AG / (c)Copyright 2023
   // ------------------------------------------------------------------------------
   // Title:            CallEnEffMonitor (FC32)
   // Comment/Function: Call of Demo EnergyMeter and Energy Efficient M for EEMM demonstration
   // Library/Family:   Energy
   // Author:           SICAR
   // Tested with:      ---
   // Engineering:      TIA Portal V19
   // Restrictions:     -
   // Requirements:     ---
   // ------------------------------------------------------------------------------
   // Change log table:
   // Version  | Date       | Expert in charge       | Changes applied
   // ---------|------------|------------------------|------------------------------
   // 05.00.00 | 01.09.2023 | SICAR
   //                         First released version
END_REGION

